C09100=1019.861,101.441,387.765,167.239,51.912,159.574
C09101=1019.866,101.689,387.746,167.241,51.905,159.573
C09102=1019.872,101.938,387.728,167.244,51.898,159.572
C09103=1019.877,102.188,387.710,167.246,51.892,159.571
C09104=1019.882,102.438,387.692,167.249,51.885,159.571
C09105=1019.888,102.686,387.673,167.252,51.878,159.570
C09106=1019.893,102.936,387.655,167.255,51.871,159.569
C09107=1019.898,103.185,387.637,167.257,51.864,159.568
C09108=1019.903,103.435,387.619,167.260,51.857,159.567
C09109=1019.910,103.684,387.601,167.263,51.851,159.567
C09110=1019.914,103.933,387.582,167.266,51.844,159.566
C09111=1019.919,104.182,387.564,167.269,51.838,159.565
C09112=1019.925,104.432,387.546,167.272,51.831,159.564
C09113=1019.930,104.681,387.527,167.274,51.824,159.563
C09114=1019.936,104.930,387.510,167.277,51.817,159.563
C09115=1019.941,105.180,387.491,167.280,51.811,159.562
C09116=1019.946,105.429,387.472,167.283,51.804,159.561
C09117=1019.952,105.678,387.455,167.285,51.797,159.560
C09118=1019.957,105.928,387.436,167.288,51.790,159.559
C09119=1019.963,106.176,387.418,167.292,51.783,159.559
C09120=1019.968,106.426,387.400,167.294,51.776,159.558
C09121=1019.974,106.675,387.382,167.297,51.769,159.557
C09122=1019.979,106.958,387.360,167.300,51.762,159.556
C09123=1019.986,107.241,387.340,167.303,51.754,159.555
C09124=1019.992,107.524,387.319,167.307,51.746,159.554
C09125=1019.998,107.806,387.298,167.310,51.738,159.553
C09126=1020.004,108.056,387.280,167.312,51.732,159.552
C09127=1020.009,108.305,387.262,167.315,51.725,159.551
C09128=1020.014,108.554,387.243,167.318,51.718,159.551
C09129=1020.020,108.804,387.225,167.321,51.711,159.550
C09130=1020.025,109.052,387.206,167.324,51.704,159.549
C09131=1020.032,109.302,387.188,167.326,51.698,159.548
C09132=1020.036,109.551,387.170,167.330,51.691,159.547
C09133=1020.041,109.800,387.151,167.332,51.684,159.546
C09134=1020.047,110.050,387.133,167.335,51.678,159.546
C09135=1020.053,110.299,387.115,167.338,51.671,159.545
C09136=1020.058,110.549,387.096,167.341,51.664,159.544
C09137=1020.063,110.797,387.077,167.344,51.657,159.543
C09138=1020.068,111.047,387.059,167.347,51.651,159.543
C09139=1020.074,111.296,387.040,167.350,51.644,159.542
C09140=1020.079,111.545,387.021,167.352,51.637,159.541
C09141=1020.085,111.795,387.003,167.355,51.630,159.540
C09142=1020.090,112.043,386.984,167.358,51.623,159.539
C09143=1020.095,112.293,386.966,167.361,51.616,159.539
C09144=1020.100,112.542,386.947,167.363,51.610,159.538
C09145=1020.106,112.792,386.927,167.367,51.603,159.537
C09146=1020.111,113.041,386.909,167.369,51.597,159.536
C09147=1020.116,113.290,386.890,167.373,51.590,159.535
C09148=1020.122,113.539,386.871,167.375,51.583,159.535
C09149=1020.127,113.789,386.853,167.378,51.576,159.534
C09150=1020.132,114.038,386.834,167.380,51.570,159.533
C09151=1020.137,114.287,386.815,167.384,51.564,159.532
C09152=1020.143,114.536,386.796,167.386,51.557,159.531
C09153=1020.148,114.785,386.777,167.390,51.550,159.531
C09154=1020.153,115.035,386.758,167.392,51.543,159.530
C09155=1020.158,115.284,386.739,167.395,51.536,159.529
C09156=1020.164,115.533,386.720,167.398,51.530,159.528
C09157=1020.169,115.782,386.702,167.401,51.523,159.527
C09158=1020.175,116.032,386.683,167.404,51.517,159.527
C09159=1020.179,116.281,386.663,167.407,51.510,159.526
C09160=1020.185,116.530,386.644,167.409,51.504,159.525
C09161=1020.190,116.779,386.625,167.412,51.497,159.524
C09162=1020.195,117.029,386.607,167.415,51.490,159.523
C09163=1020.200,117.278,386.588,167.418,51.483,159.523
C09164=1020.206,117.527,386.568,167.421,51.476,159.522
C09165=1020.211,117.776,386.550,167.424,51.470,159.521
C09166=1020.217,118.025,386.530,167.427,51.463,159.520
C09167=1020.222,118.274,386.511,167.430,51.457,159.520
C09168=1020.227,118.524,386.493,167.433,51.450,159.519
C09169=1020.232,118.773,386.474,167.435,51.443,159.518
C09170=1020.238,119.022,386.455,167.439,51.436,159.517
C09171=1020.243,119.271,386.436,167.441,51.430,159.516
C09172=1020.249,119.521,386.417,167.444,51.423,159.516
C09173=1020.254,119.770,386.397,167.448,51.416,159.515
C09174=1020.259,120.019,386.378,167.450,51.409,159.514
C09175=1020.264,120.268,386.359,167.454,51.403,159.513
C09176=1020.269,120.517,386.340,167.456,51.396,159.512
C09177=1020.275,120.767,386.321,167.459,51.390,159.512
C09178=1020.280,121.016,386.302,167.463,51.383,159.511
C09179=1020.286,121.265,386.283,167.465,51.376,159.510
C09180=1020.291,121.515,386.264,167.468,51.369,159.509
C09181=1020.296,121.764,386.245,167.471,51.363,159.508
C09182=1020.302,122.013,386.226,167.474,51.356,159.508
C09183=1020.307,122.262,386.207,167.477,51.349,159.507
C09184=1020.313,122.511,386.188,167.480,51.342,159.506
C09185=1020.318,122.761,386.168,167.483,51.335,159.505
C09186=1020.324,123.043,386.147,167.486,51.328,159.504
C09187=1020.330,123.326,386.125,167.490,51.320,159.503
C09188=1020.336,123.609,386.103,167.493,51.312,159.502
C09189=1020.342,123.891,386.082,167.496,51.305,159.502
C09190=1020.348,124.141,386.062,167.499,51.298,159.501
C09191=1020.353,124.389,386.043,167.503,51.291,159.500
C09192=1020.359,124.639,386.024,167.505,51.285,159.499
C09193=1020.364,124.889,386.004,167.508,51.278,159.498
C09194=1020.369,125.137,385.985,167.512,51.271,159.498
C09195=1020.375,125.387,385.966,167.514,51.264,159.497
C09196=1020.380,125.636,385.947,167.517,51.257,159.496
C09197=1020.385,125.885,385.928,167.520,51.251,159.495
C09198=1020.391,126.134,385.909,167.523,51.244,159.494
C09199=1020.397,126.384,385.890,167.526,51.237,159.494
C09200=1020.402,126.633,385.871,167.530,51.230,159.493
C09201=1020.408,126.882,385.852,167.532,51.224,159.492
C09202=1020.413,127.131,385.832,167.536,51.217,159.491
C09203=1020.418,127.380,385.812,167.539,51.210,159.490
C09204=1020.424,127.629,385.793,167.541,51.203,159.489
C09205=1020.429,127.879,385.774,167.544,51.196,159.489
C09206=1020.435,128.128,385.754,167.548,51.189,159.488
C09207=1020.440,128.377,385.735,167.550,51.182,159.487
C09208=1020.446,128.626,385.716,167.553,51.175,159.486
C09209=1020.451,128.876,385.697,167.557,51.169,159.485
C09210=1020.456,129.124,385.678,167.559,51.162,159.484
C09211=1020.462,129.374,385.659,167.562,51.155,159.484
C09212=1020.468,129.623,385.639,167.566,51.148,159.483
C09213=1020.473,129.872,385.619,167.569,51.141,159.482
C09214=1020.478,130.121,385.600,167.571,51.135,159.481
C09215=1020.484,130.371,385.581,167.575,51.128,159.481
C09216=1020.489,130.620,385.560,167.577,51.122,159.480
C09217=1020.495,130.869,385.541,167.581,51.115,159.479
C09218=1020.500,131.119,385.521,167.584,51.108,159.478
C09219=1020.505,131.368,385.502,167.587,51.102,159.477
C09220=1020.510,131.617,385.482,167.590,51.095,159.477
C09221=1020.516,131.866,385.463,167.593,51.088,159.476
C09222=1020.520,132.115,385.442,167.596,51.082,159.475
C09223=1020.526,132.364,385.423,167.599,51.075,159.474
C09224=1020.532,132.614,385.404,167.603,51.068,159.474
C09225=1020.537,132.863,385.383,167.605,51.062,159.473
C09226=1020.543,133.112,385.364,167.609,51.055,159.472
C09227=1020.547,133.361,385.345,167.611,51.049,159.471
C09228=1020.553,133.610,385.325,167.614,51.042,159.470
C09229=1020.558,133.860,385.305,167.618,51.035,159.470
C09230=1020.564,134.108,385.285,167.620,51.028,159.469
C09231=1020.568,134.358,385.265,167.623,51.021,159.468
C09232=1020.574,134.606,385.246,167.627,51.015,159.467
C09233=1020.579,134.856,385.226,167.630,51.008,159.466
C09234=1020.585,135.106,385.206,167.633,51.001,159.466
C09235=1020.591,135.354,385.186,167.636,50.995,159.465
C09236=1020.595,135.603,385.167,167.640,50.988,159.464
C09237=1020.601,135.852,385.147,167.642,50.982,159.463
C09238=1020.606,136.102,385.127,167.645,50.975,159.463
C09239=1020.612,136.351,385.107,167.649,50.968,159.462
C09240=1020.617,136.600,385.087,167.651,50.961,159.461
C09241=1020.623,136.850,385.067,167.655,50.955,159.460
C09242=1020.628,137.098,385.048,167.658,50.948,159.459
C09243=1020.633,137.347,385.027,167.660,50.941,159.459
C09244=1020.639,137.596,385.007,167.664,50.934,159.458
C09245=1020.644,137.846,384.988,167.668,50.928,159.457
C09246=1020.650,138.095,384.968,167.671,50.921,159.456
C09247=1020.655,138.345,384.948,167.673,50.915,159.456
C09248=1020.659,138.593,384.928,167.677,50.908,159.455
C09249=1020.665,138.842,384.908,167.680,50.901,159.454
C09250=1020.671,139.125,384.885,167.683,50.894,159.453
C09251=1020.677,139.408,384.862,167.687,50.887,159.452
C09252=1020.684,139.690,384.839,167.691,50.879,159.451
C09253=1020.689,139.973,384.816,167.694,50.871,159.450
C09254=1020.695,140.222,384.796,167.697,50.864,159.450
C09255=1020.700,140.472,384.776,167.701,50.858,159.449
C09256=1020.705,140.720,384.756,167.703,50.852,159.448
C09257=1020.710,140.969,384.736,167.707,50.845,159.447
C09258=1020.716,141.219,384.716,167.710,50.838,159.447
C09259=1020.721,141.468,384.696,167.712,50.832,159.446
C09260=1020.726,141.717,384.675,167.716,50.825,159.445
C09261=1020.732,141.966,384.655,167.719,50.818,159.444
C09262=1020.737,142.215,384.635,167.723,50.812,159.444
C09263=1020.743,142.464,384.615,167.725,50.805,159.443
C09264=1020.748,142.714,384.594,167.729,50.799,159.442
C09265=1020.754,142.962,384.574,167.732,50.792,159.441
C09266=1020.759,143.212,384.555,167.735,50.785,159.440
C09267=1020.763,143.461,384.534,167.738,50.778,159.440
C09268=1020.769,143.710,384.514,167.742,50.772,159.439
C09269=1020.775,143.959,384.494,167.745,50.765,159.438
C09270=1020.780,144.208,384.473,167.748,50.759,159.437
C09271=1020.785,144.457,384.453,167.751,50.752,159.437
C09272=1020.790,144.707,384.433,167.755,50.745,159.436
C09273=1020.796,144.955,384.413,167.758,50.738,159.435
C09274=1020.801,145.204,384.392,167.760,50.732,159.434
C09275=1020.807,145.454,384.372,167.764,50.725,159.433
C09276=1020.813,145.702,384.352,167.767,50.718,159.433
C09277=1020.818,145.952,384.331,167.771,50.712,159.432
C09278=1020.823,146.201,384.311,167.774,50.706,159.431
C09279=1020.828,146.450,384.290,167.777,50.699,159.430
C09280=1020.834,146.699,384.270,167.780,50.692,159.430
C09281=1020.839,146.949,384.250,167.784,50.685,159.429
C09282=1020.844,147.198,384.229,167.787,50.680,159.428
C09283=1020.849,147.447,384.209,167.790,50.673,159.427
C09284=1020.854,147.696,384.188,167.794,50.666,159.427
C09285=1020.860,147.945,384.168,167.797,50.659,159.426
C09286=1020.865,148.194,384.146,167.800,50.653,159.425
C09287=1020.870,148.443,384.126,167.803,50.647,159.424
C09288=1020.876,148.692,384.105,167.807,50.640,159.424
C09289=1020.881,148.941,384.085,167.810,50.633,159.423
C09290=1020.886,149.190,384.064,167.812,50.626,159.422
C09291=1020.891,149.439,384.044,167.816,50.620,159.421
C09292=1020.897,149.688,384.023,167.820,50.614,159.421
C09293=1020.902,149.938,384.002,167.823,50.607,159.420
C09294=1020.907,150.187,383.982,167.826,50.600,159.419
C09295=1020.912,150.436,383.961,167.829,50.594,159.418
C09296=1020.918,150.685,383.941,167.833,50.587,159.418
C09297=1020.923,150.934,383.920,167.836,50.581,159.417
C09298=1020.929,151.183,383.899,167.839,50.574,159.416
C09299=1020.934,151.432,383.878,167.842,50.567,159.415
C09300=1020.940,151.681,383.858,167.846,50.561,159.415
C09301=1020.945,151.931,383.837,167.850,50.554,159.414
C09302=1020.950,152.180,383.816,167.853,50.548,159.413
C09303=1020.955,152.429,383.796,167.855,50.541,159.412
C09304=1020.961,152.677,383.775,167.859,50.534,159.411
C09305=1020.966,152.926,383.754,167.863,50.528,159.411
C09306=1020.971,153.176,383.733,167.866,50.522,159.410
C09307=1020.977,153.425,383.713,167.870,50.515,159.409
C09308=1020.982,153.674,383.692,167.872,50.508,159.408
C09309=1020.988,153.923,383.671,167.876,50.502,159.408
C09310=1020.993,154.172,383.650,167.879,50.495,159.407
C09311=1020.999,154.421,383.630,167.883,50.489,159.406
C09312=1021.003,154.670,383.608,167.887,50.483,159.406
C09313=1021.009,154.919,383.587,167.889,50.476,159.405
C09314=1021.015,155.201,383.563,167.893,50.468,159.404
C09315=1021.021,155.484,383.540,167.897,50.462,159.403
C09316=1021.027,155.766,383.516,167.901,50.454,159.402
C09317=1021.033,156.050,383.493,167.905,50.446,159.402
C09318=1021.039,156.298,383.471,167.908,50.440,159.401
C09319=1021.043,156.548,383.450,167.911,50.433,159.400
C09320=1021.049,156.797,383.430,167.915,50.427,159.399
C09321=1021.054,157.045,383.408,167.918,50.420,159.399
C09322=1021.059,157.294,383.388,167.922,50.414,159.398
C09323=1021.066,157.543,383.366,167.926,50.407,159.397
C09324=1021.071,157.793,383.346,167.928,50.401,159.396
C09325=1021.075,158.042,383.324,167.931,50.394,159.396
C09326=1021.081,158.291,383.303,167.935,50.388,159.395
C09327=1021.086,158.540,383.283,167.939,50.381,159.394
C09328=1021.092,158.789,383.261,167.942,50.374,159.393
C09329=1021.098,159.038,383.240,167.946,50.368,159.393
C09330=1021.102,159.287,383.219,167.949,50.362,159.392
C09331=1021.107,159.536,383.197,167.952,50.356,159.391
C09332=1021.113,159.785,383.176,167.956,50.349,159.391
C09333=1021.117,160.034,383.154,167.959,50.342,159.390
C09334=1021.123,160.283,383.132,167.962,50.337,159.389
C09335=1021.128,160.532,383.112,167.966,50.330,159.388
C09336=1021.133,160.781,383.090,167.970,50.324,159.388
C09337=1021.138,161.030,383.068,167.973,50.317,159.387
C09338=1021.143,161.279,383.047,167.976,50.311,159.386
C09339=1021.148,161.528,383.025,167.979,50.304,159.386
C09340=1021.154,161.777,383.004,167.983,50.298,159.385
C09341=1021.159,162.026,382.982,167.987,50.292,159.384
C09342=1021.163,162.275,382.961,167.991,50.286,159.384
C09343=1021.169,162.524,382.939,167.993,50.279,159.383
C09344=1021.174,162.773,382.917,167.997,50.273,159.382
C09345=1021.180,163.022,382.896,168.000,50.266,159.381
C09346=1021.184,163.271,382.875,168.004,50.260,159.381
C09347=1021.189,163.520,382.853,168.008,50.254,159.380
C09348=1021.195,163.769,382.831,168.011,50.248,159.379
C09349=1021.200,164.018,382.809,168.014,50.241,159.379
C09350=1021.205,164.267,382.788,168.018,50.235,159.378
C09351=1021.211,164.517,382.767,168.022,50.228,159.377
C09352=1021.216,164.765,382.745,168.025,50.222,159.377
C09353=1021.221,165.014,382.723,168.028,50.216,159.376
C09354=1021.226,165.263,382.702,168.031,50.209,159.375
C09355=1021.231,165.512,382.679,168.035,50.203,159.374
C09356=1021.237,165.761,382.658,168.039,50.196,159.374
C09357=1021.242,166.010,382.637,168.043,50.190,159.373
C09358=1021.247,166.260,382.615,168.046,50.184,159.372
C09359=1021.253,166.508,382.594,168.050,50.178,159.372
C09360=1021.257,166.757,382.572,168.053,50.171,159.371
C09361=1021.263,167.007,382.549,168.056,50.165,159.370
C09362=1021.268,167.255,382.528,168.060,50.158,159.370
C09363=1021.273,167.504,382.506,168.064,50.152,159.369
C09364=1021.279,167.753,382.484,168.067,50.146,159.368
C09365=1021.284,168.002,382.463,168.071,50.140,159.368
C09366=1021.289,168.251,382.441,168.075,50.133,159.367
C09367=1021.294,168.500,382.419,168.078,50.126,159.366
C09368=1021.300,168.749,382.397,168.082,50.120,159.365
C09369=1021.305,168.998,382.376,168.085,50.114,159.365
C09370=1021.311,169.247,382.355,168.089,50.108,159.364
C09371=1021.315,169.496,382.333,168.092,50.101,159.363
C09372=1021.321,169.746,382.311,168.096,50.095,159.363
C09373=1021.326,169.994,382.289,168.100,50.088,159.362
C09374=1021.331,170.243,382.267,168.103,50.082,159.361
C09375=1021.337,170.493,382.245,168.107,50.076,159.360
C09376=1021.342,170.741,382.224,168.111,50.070,159.360
C09377=1021.348,170.990,382.201,168.114,50.063,159.359
C09378=1021.354,171.272,382.177,168.119,50.056,159.358
C09379=1021.360,171.554,382.151,168.122,50.048,159.357
C09380=1021.366,171.836,382.127,168.127,50.041,159.357
C09381=1021.372,172.118,382.102,168.131,50.034,159.356
C09382=1021.377,172.367,382.080,168.135,50.028,159.355
C09383=1021.383,172.617,382.058,168.138,50.021,159.355
C09384=1021.388,172.865,382.037,168.142,50.015,159.354
C09385=1021.394,173.115,382.015,168.146,50.008,159.353
C09386=1021.398,173.364,381.993,168.150,50.002,159.353
C09387=1021.405,173.613,381.971,168.153,49.996,159.352
C09388=1021.409,173.862,381.949,168.157,49.989,159.351
C09389=1021.415,174.111,381.926,168.161,49.983,159.350
C09390=1021.421,174.359,381.905,168.164,49.976,159.350
C09391=1021.426,174.609,381.883,168.168,49.970,159.349
C09392=1021.431,174.857,381.861,168.171,49.964,159.348
C09393=1021.437,175.107,381.839,168.175,49.957,159.348
C09394=1021.442,175.355,381.817,168.179,49.951,159.347
C09395=1021.448,175.604,381.795,168.183,49.945,159.346
C09396=1021.453,175.853,381.773,168.186,49.938,159.346
C09397=1021.459,176.102,381.751,168.190,49.931,159.345
C09398=1021.464,176.352,381.729,168.194,49.925,159.344
C09399=1021.470,176.600,381.707,168.197,49.919,159.343
C09400=1021.475,176.849,381.685,168.201,49.913,159.343
C09401=1021.480,177.098,381.663,168.205,49.906,159.342
C09402=1021.486,177.347,381.641,168.209,49.900,159.341
C09403=1021.492,177.595,381.619,168.212,49.893,159.341
C09404=1021.497,177.845,381.596,168.216,49.887,159.340
C09405=1021.502,178.095,381.574,168.220,49.881,159.339
C09406=1021.508,178.343,381.553,168.223,49.874,159.339
C09407=1021.514,178.592,381.530,168.227,49.868,159.338
C09408=1021.518,178.841,381.508,168.231,49.861,159.337
C09409=1021.525,179.090,381.486,168.236,49.855,159.337
C09410=1021.530,179.339,381.463,168.239,49.848,159.336
C09411=1021.535,179.588,381.442,168.243,49.842,159.335
C09412=1021.541,179.837,381.420,168.247,49.836,159.335
C09413=1021.547,180.086,381.397,168.251,49.830,159.334
C09414=1021.552,180.335,381.375,168.254,49.823,159.333
C09415=1021.558,180.584,381.353,168.258,49.817,159.333
C09416=1021.564,180.833,381.331,168.262,49.810,159.332
C09417=1021.569,181.081,381.309,168.265,49.804,159.331
C09418=1021.575,181.330,381.286,168.270,49.798,159.331
C09419=1021.581,181.580,381.264,168.274,49.791,159.330
C09420=1021.586,181.828,381.241,168.278,49.785,159.329
C09421=1021.591,182.077,381.219,168.281,49.778,159.328
C09422=1021.597,182.327,381.197,168.285,49.772,159.328
C09423=1021.602,182.575,381.174,168.289,49.766,159.327
C09424=1021.607,182.824,381.152,168.293,49.760,159.326
C09425=1021.612,183.074,381.129,168.297,49.754,159.326
C09426=1021.618,183.323,381.106,168.301,49.748,159.325
C09427=1021.623,183.571,381.083,168.305,49.742,159.325
C09428=1021.628,183.820,381.060,168.308,49.736,159.324
C09429=1021.633,184.070,381.037,168.312,49.729,159.323
C09430=1021.638,184.318,381.015,168.316,49.723,159.323
C09431=1021.644,184.567,380.992,168.320,49.717,159.322
C09432=1021.649,184.816,380.968,168.324,49.711,159.322
C09433=1021.654,185.064,380.946,168.327,49.705,159.321
C09434=1021.660,185.314,380.924,168.331,49.699,159.320
C09435=1021.665,185.563,380.900,168.335,49.693,159.320
C09436=1021.670,185.811,380.877,168.339,49.687,159.319
C09437=1021.676,186.060,380.854,168.343,49.681,159.318
C09438=1021.681,186.309,380.831,168.347,49.674,159.318
C09439=1021.686,186.558,380.808,168.351,49.668,159.317
C09440=1021.691,186.806,380.785,168.355,49.662,159.316
C09441=1021.696,187.056,380.763,168.359,49.656,159.316
C09442=1021.702,187.338,380.736,168.363,49.649,159.315
C09443=1021.708,187.619,380.710,168.368,49.642,159.314
C09444=1021.714,187.901,380.684,168.372,49.635,159.314
C09445=1021.720,188.183,380.658,168.377,49.628,159.313
C09446=1021.726,188.431,380.636,168.381,49.622,159.312
C09447=1021.731,188.680,380.613,168.385,49.616,159.312
C09448=1021.736,188.929,380.589,168.388,49.610,159.311
C09449=1021.742,189.178,380.566,168.392,49.604,159.310
C09450=1021.748,189.427,380.543,168.396,49.598,159.310
C09451=1021.752,189.676,380.520,168.401,49.591,159.309
C09452=1021.758,189.924,380.497,168.405,49.585,159.309
C09453=1021.764,190.173,380.474,168.409,49.579,159.308
C09454=1021.769,190.423,380.451,168.413,49.573,159.307
C09455=1021.774,190.671,380.428,168.417,49.567,159.307
C09456=1021.780,190.920,380.405,168.420,49.561,159.306
C09457=1021.784,191.169,380.381,168.424,49.555,159.305
C09458=1021.790,191.418,380.359,168.429,49.549,159.305
C09459=1021.796,191.667,380.336,168.433,49.543,159.304
C09460=1021.801,191.916,380.312,168.437,49.537,159.304
C09461=1021.807,192.165,380.289,168.441,49.531,159.303
C09462=1021.813,192.413,380.265,168.445,49.524,159.302
C09463=1021.818,192.662,380.242,168.449,49.518,159.302
C09464=1021.823,192.911,380.219,168.454,49.512,159.301
C09465=1021.828,193.160,380.196,168.458,49.506,159.301
C09466=1021.834,193.409,380.173,168.462,49.500,159.300
C09467=1021.839,193.657,380.150,168.465,49.493,159.299
C09468=1021.844,193.907,380.126,168.469,49.488,159.299
C09469=1021.850,194.156,380.103,168.474,49.481,159.298
C09470=1021.856,194.404,380.080,168.478,49.475,159.298
C09471=1021.861,194.653,380.056,168.482,49.469,159.297
C09472=1021.867,194.902,380.033,168.486,49.464,159.296
C09473=1021.872,195.151,380.010,168.490,49.457,159.296
C09474=1021.877,195.400,379.987,168.495,49.451,159.295
C09475=1021.883,195.648,379.963,168.499,49.445,159.295
C09476=1021.889,195.897,379.940,168.503,49.439,159.294
C09477=1021.894,196.146,379.917,168.507,49.433,159.293
C09478=1021.900,196.395,379.894,168.512,49.427,159.293
C09479=1021.905,196.644,379.869,168.516,49.421,159.292
C09480=1021.911,196.893,379.846,168.519,49.414,159.291
C09481=1021.917,197.142,379.824,168.523,49.408,159.291
C09482=1021.922,197.390,379.799,168.528,49.402,159.290
C09483=1021.928,197.639,379.776,168.532,49.396,159.290
C09484=1021.933,197.888,379.753,168.536,49.390,159.289
C09485=1021.939,198.137,379.729,168.540,49.384,159.289
C09486=1021.944,198.386,379.706,168.545,49.378,159.288
C09487=1021.950,198.634,379.683,168.549,49.372,159.287
C09488=1021.956,198.883,379.659,168.553,49.366,159.287
C09489=1021.961,199.132,379.636,168.558,49.359,159.286
C09490=1021.966,199.381,379.613,168.562,49.354,159.286
C09491=1021.972,199.629,379.589,168.566,49.348,159.285
C09492=1021.977,199.879,379.565,168.571,49.341,159.284
C09493=1021.984,200.128,379.541,168.575,49.336,159.284
C09494=1021.989,200.377,379.518,168.579,49.330,159.283
C09495=1021.994,200.625,379.493,168.583,49.324,159.283
C09496=1021.999,200.874,379.469,168.586,49.318,159.282
C09497=1022.005,201.123,379.446,168.591,49.312,159.281
C09498=1022.011,201.371,379.422,168.595,49.306,159.281
C09499=1022.016,201.621,379.398,168.599,49.300,159.280
C09500=1022.021,201.869,379.374,168.604,49.294,159.280
C09501=1022.027,202.118,379.351,168.608,49.288,159.279
C09502=1022.032,202.367,379.327,168.613,49.283,159.279
C09503=1022.037,202.615,379.303,168.617,49.277,159.278
C09504=1022.043,202.865,379.278,168.622,49.270,159.278
C09505=1022.049,203.114,379.255,168.626,49.265,159.277
C09506=1022.077,204.361,379.134,169.059,49.356,159.363
C09507=1022.082,204.574,379.111,169.061,49.352,159.363
C09508=1022.088,204.787,379.090,169.065,49.348,159.363
C09509=1022.093,205.000,379.068,169.067,49.343,159.362
C09510=1022.099,205.213,379.046,169.071,49.339,159.362
C09511=1022.104,205.425,379.025,169.073,49.334,159.361
C09512=1022.109,205.639,379.002,169.077,49.330,159.361
C09513=1022.115,205.852,378.981,169.079,49.326,159.360
C09514=1022.121,206.100,378.955,169.083,49.321,159.360
C09515=1022.128,206.349,378.929,169.086,49.317,159.359
C09516=1022.134,206.598,378.904,169.089,49.312,159.359
C09517=1022.141,206.846,378.878,169.093,49.307,159.358
C09518=1022.147,207.095,378.853,169.096,49.302,159.358
C09519=1022.153,207.343,378.827,169.100,49.297,159.357
C09520=1022.159,207.592,378.802,169.103,49.292,159.357
C09521=1022.166,207.840,378.776,169.107,49.287,159.356
C09522=1022.171,208.089,378.750,169.110,49.282,159.356
C09523=1022.178,208.339,378.724,169.113,49.277,159.355
C09524=1022.185,208.587,378.698,169.117,49.272,159.355
C09525=1022.191,208.835,378.673,169.120,49.267,159.354
C09526=1022.197,209.083,378.647,169.123,49.262,159.353
C09527=1022.203,209.332,378.621,169.127,49.258,159.353
C09528=1022.210,209.581,378.596,169.130,49.253,159.352
C09529=1022.216,209.830,378.569,169.134,49.248,159.352
C09530=1022.222,210.078,378.544,169.138,49.243,159.352
C09531=1022.229,210.326,378.518,169.141,49.238,159.351
C09532=1022.235,210.575,378.492,169.144,49.234,159.351
C09533=1022.241,210.823,378.466,169.148,49.229,159.350
C09534=1022.247,211.072,378.440,169.151,49.224,159.349
C09535=1022.254,211.321,378.414,169.155,49.220,159.349
C09536=1022.260,211.570,378.388,169.158,49.215,159.349
C09537=1022.266,211.818,378.362,169.161,49.210,159.348
C09538=1022.272,212.067,378.337,169.164,49.205,159.348
C09539=1022.278,212.315,378.310,169.168,49.201,159.347
C09540=1022.285,212.564,378.284,169.171,49.196,159.347
C09541=1022.291,212.812,378.258,169.175,49.191,159.346
C09542=1022.297,213.061,378.232,169.178,49.187,159.346
C09543=1022.303,213.309,378.206,169.182,49.182,159.345
C09544=1022.310,213.558,378.180,169.185,49.177,159.345
C09545=1022.316,213.807,378.154,169.190,49.172,159.344
C09546=1022.322,214.055,378.128,169.193,49.168,159.344
C09547=1022.329,214.303,378.102,169.196,49.163,159.343
C09548=1022.335,214.553,378.076,169.200,49.158,159.343
C09549=1022.342,214.801,378.049,169.203,49.154,159.343
C09550=1022.348,215.049,378.023,169.206,49.149,159.342
C09551=1022.354,215.299,377.997,169.210,49.145,159.342
C09552=1022.361,215.547,377.971,169.213,49.140,159.341
C09553=1022.367,215.795,377.945,169.217,49.135,159.341
C09554=1022.373,216.044,377.919,169.220,49.131,159.340
C09555=1022.380,216.292,377.893,169.224,49.126,159.340
C09556=1022.386,216.541,377.867,169.227,49.121,159.339
C09557=1022.392,216.789,377.840,169.231,49.117,159.339
C09558=1022.399,217.038,377.814,169.234,49.112,159.338
C09559=1022.405,217.287,377.788,169.238,49.108,159.338
C09560=1022.411,217.535,377.762,169.241,49.103,159.337
C09561=1022.418,217.783,377.735,169.245,49.098,159.337
C09562=1022.424,218.032,377.709,169.249,49.093,159.337
C09563=1022.430,218.280,377.683,169.252,49.089,159.336
C09564=1022.437,218.529,377.657,169.256,49.084,159.336
C09565=1022.443,218.778,377.630,169.259,49.080,159.335
C09566=1022.449,218.993,377.607,169.262,49.076,159.335
C09567=1022.454,219.207,377.585,169.265,49.072,159.334
C09568=1022.460,219.422,377.561,169.269,49.068,159.334
C09569=1022.464,219.637,377.538,169.271,49.064,159.334
C09570=1022.470,219.852,377.516,169.274,49.060,159.333
C09571=1022.475,220.067,377.493,169.278,49.057,159.333
C09572=1022.481,220.281,377.470,169.280,49.053,159.333
C09573=1022.486,220.496,377.447,169.283,49.049,159.332
C09574=1022.493,220.745,377.420,169.287,49.045,159.332
C09575=1022.499,220.993,377.394,169.290,49.040,159.331
C09576=1022.505,221.241,377.367,169.294,49.036,159.331
C09577=1022.512,221.490,377.341,169.297,49.032,159.331
C09578=1022.517,221.739,377.314,169.301,49.027,159.330
C09579=1022.525,221.987,377.288,169.304,49.023,159.330
C09580=1022.530,222.236,377.261,169.308,49.018,159.329
C09581=1022.536,222.484,377.234,169.311,49.014,159.329
C09582=1022.543,222.733,377.208,169.315,49.009,159.329
C09583=1022.549,222.981,377.181,169.319,49.005,159.328
C09584=1022.555,223.230,377.154,169.322,49.000,159.328
C09585=1022.562,223.478,377.128,169.326,48.996,159.327
C09586=1022.568,223.727,377.101,169.329,48.992,159.327
C09587=1022.574,223.975,377.074,169.333,48.988,159.327
C09588=1022.581,224.224,377.047,169.336,48.983,159.326
C09589=1022.587,224.472,377.021,169.340,48.979,159.326
C09590=1022.593,224.721,376.994,169.344,48.975,159.325
C09591=1022.600,224.969,376.968,169.347,48.970,159.325
C09592=1022.606,225.218,376.941,169.351,48.966,159.324
C09593=1022.612,225.467,376.914,169.354,48.961,159.324
C09594=1022.619,225.714,376.887,169.358,48.957,159.324
C09595=1022.625,225.963,376.860,169.362,48.953,159.323
C09596=1022.631,226.212,376.834,169.366,48.949,159.323
C09597=1022.638,226.460,376.807,169.370,48.944,159.323
C09598=1022.644,226.709,376.780,169.373,48.940,159.322
C09599=1022.652,226.957,376.753,169.377,48.935,159.322
C09600=1022.657,227.205,376.727,169.381,48.931,159.322
C09601=1022.664,227.454,376.700,169.383,48.927,159.321
C09602=1022.670,227.702,376.672,169.387,48.923,159.321
C09603=1022.676,227.951,376.645,169.391,48.919,159.320
C09604=1022.682,228.199,376.619,169.394,48.915,159.320
C09605=1022.689,228.448,376.591,169.398,48.911,159.320
C09606=1022.695,228.697,376.564,169.402,48.907,159.319
C09607=1022.701,228.945,376.537,169.405,48.902,159.319
C09608=1022.707,229.194,376.510,169.409,48.898,159.319
C09609=1022.714,229.442,376.483,169.413,48.894,159.318
C09610=1022.721,229.690,376.456,169.416,48.890,159.318
C09611=1022.726,229.939,376.429,169.420,48.886,159.318
C09612=1022.733,230.188,376.402,169.424,48.882,159.317
C09613=1022.739,230.435,376.375,169.427,48.877,159.317
C09614=1022.745,230.684,376.348,169.431,48.873,159.317
C09615=1022.752,230.933,376.320,169.435,48.869,159.316
C09616=1022.758,231.181,376.293,169.438,48.865,159.316
C09617=1022.764,231.430,376.266,169.442,48.861,159.315
C09618=1022.770,231.677,376.238,169.446,48.857,159.315
C09619=1022.777,231.926,376.211,169.449,48.852,159.315
C09620=1022.783,232.175,376.183,169.453,48.849,159.315
C09621=1022.789,232.423,376.157,169.457,48.845,159.314
C09622=1022.795,232.672,376.128,169.461,48.841,159.314
C09623=1022.801,232.920,376.102,169.465,48.836,159.314
C09624=1022.808,233.169,376.074,169.468,48.832,159.313
C09625=1022.814,233.417,376.046,169.471,48.828,159.313
C09626=1022.824,233.793,376.006,169.477,48.823,159.312
C09627=1022.834,234.169,375.964,169.482,48.817,159.312
C09628=1022.843,234.546,375.923,169.488,48.810,159.311
C09629=1022.853,234.922,375.881,169.494,48.805,159.311
C09630=1022.859,235.170,375.854,169.497,48.801,159.311
C09631=1022.865,235.419,375.826,169.501,48.796,159.310
C09632=1022.872,235.667,375.799,169.505,48.792,159.310
C09633=1022.878,235.915,375.771,169.509,48.789,159.310
C09634=1022.884,236.165,375.744,169.512,48.785,159.309
C09635=1022.891,236.413,375.716,169.516,48.780,159.309
C09636=1022.897,236.661,375.689,169.520,48.776,159.309
C09637=1022.903,236.909,375.661,169.524,48.773,159.309
C09638=1022.910,237.158,375.633,169.527,48.769,159.308
C09639=1022.916,237.407,375.606,169.531,48.765,159.308
C09640=1022.922,237.654,375.579,169.535,48.761,159.308
C09641=1022.929,237.903,375.551,169.539,48.757,159.307
C09642=1022.935,238.152,375.523,169.543,48.753,159.307
C09643=1022.942,238.400,375.495,169.547,48.749,159.307
C09644=1022.948,238.648,375.468,169.550,48.745,159.306
C09645=1022.954,238.897,375.441,169.554,48.741,159.306
C09646=1022.961,239.145,375.413,169.558,48.737,159.306
C09647=1022.968,239.394,375.385,169.562,48.733,159.306
C09648=1022.973,239.642,375.357,169.566,48.730,159.305
C09649=1022.980,239.890,375.330,169.569,48.726,159.305
C09650=1022.986,240.139,375.302,169.572,48.722,159.305
C09651=1022.992,240.387,375.273,169.576,48.718,159.304
C09652=1022.998,240.635,375.246,169.580,48.715,159.304
C09653=1023.004,240.884,375.218,169.584,48.711,159.304
C09654=1023.011,241.132,375.190,169.588,48.707,159.304
C09655=1023.018,241.380,375.162,169.592,48.704,159.304
C09656=1023.023,241.628,375.134,169.595,48.700,159.303
C09657=1023.030,241.877,375.106,169.600,48.696,159.303
C09658=1023.036,242.125,375.078,169.603,48.692,159.303
C09659=1023.043,242.374,375.050,169.607,48.689,159.303
C09660=1023.049,242.622,375.022,169.611,48.684,159.302
C09661=1023.055,242.871,374.994,169.614,48.681,159.302
C09662=1023.061,243.119,374.966,169.618,48.678,159.302
C09663=1023.068,243.367,374.937,169.622,48.674,159.301
C09664=1023.074,243.615,374.910,169.626,48.670,159.301
C09665=1023.080,243.864,374.881,169.630,48.667,159.301
C09666=1023.087,244.113,374.854,169.633,48.662,159.301
C09667=1023.092,244.360,374.825,169.637,48.659,159.301
C09668=1023.098,244.609,374.797,169.641,48.656,159.300
C09669=1023.105,244.857,374.769,169.646,48.652,159.300
C09670=1023.111,245.105,374.740,169.649,48.649,159.300
C09671=1023.117,245.354,374.712,169.652,48.645,159.300
C09672=1023.124,245.602,374.684,169.656,48.641,159.299
C09673=1023.130,245.850,374.655,169.660,48.638,159.299
C09674=1023.136,246.099,374.627,169.664,48.634,159.299
C09675=1023.143,246.346,374.598,169.668,48.631,159.299
C09676=1023.149,246.595,374.570,169.672,48.627,159.299
C09677=1023.154,246.844,374.542,169.676,48.623,159.298
C09678=1023.162,247.138,374.508,169.680,48.620,159.298
C09679=1023.170,247.432,374.475,169.685,48.615,159.298
C09680=1023.177,247.726,374.441,169.690,48.611,159.298
C09681=1023.184,248.019,374.407,169.694,48.606,159.297
C09682=1023.195,248.434,374.359,169.701,48.601,159.297
C09683=1023.206,248.849,374.312,169.707,48.595,159.297
C09684=1023.216,249.265,374.264,169.713,48.589,159.296
C09685=1023.226,249.680,374.216,169.720,48.584,159.296
C09686=1023.233,249.928,374.188,169.724,48.580,159.296
C09687=1023.239,250.177,374.160,169.728,48.577,159.296
C09688=1023.245,250.425,374.131,169.732,48.573,159.296
C09689=1023.251,250.674,374.102,169.736,48.570,159.295
C09690=1023.258,250.922,374.074,169.740,48.566,159.295
C09691=1023.264,251.170,374.046,169.744,48.563,159.295
C09692=1023.270,251.418,374.017,169.748,48.559,159.295
C09693=1023.277,251.666,373.988,169.752,48.556,159.295
C09694=1023.283,251.915,373.960,169.756,48.553,159.295
C09695=1023.290,252.163,373.931,169.760,48.549,159.294
C09696=1023.296,252.411,373.902,169.763,48.546,159.294
C09697=1023.303,252.660,373.874,169.767,48.542,159.294
C09698=1023.309,252.908,373.845,169.771,48.539,159.294
C09699=1023.316,253.157,373.815,169.775,48.536,159.294
C09700=1023.322,253.405,373.788,169.779,48.532,159.293
C09701=1023.329,253.653,373.759,169.783,48.529,159.293
C09702=1023.335,253.901,373.730,169.787,48.525,159.293
C09703=1023.342,254.149,373.701,169.791,48.522,159.293
C09704=1023.348,254.398,373.673,169.795,48.518,159.293
C09705=1023.354,254.646,373.644,169.799,48.515,159.293
C09706=1023.360,254.894,373.615,169.804,48.511,159.292
C09707=1023.367,255.142,373.586,169.808,48.508,159.292
C09708=1023.373,255.391,373.558,169.812,48.505,159.292
C09709=1023.380,255.640,373.529,169.816,48.502,159.292
C09710=1023.387,255.887,373.500,169.819,48.498,159.292
C09711=1023.393,256.136,373.471,169.823,48.495,159.292
C09712=1023.400,256.384,373.442,169.827,48.491,159.291
C09713=1023.406,256.632,373.413,169.831,48.488,159.291
C09714=1023.413,256.880,373.385,169.835,48.485,159.291
C09715=1023.419,257.129,373.356,169.840,48.482,159.291
C09716=1023.426,257.377,373.327,169.844,48.478,159.291
C09717=1023.432,257.625,373.298,169.848,48.475,159.291
C09718=1023.439,257.873,373.269,169.852,48.471,159.291
C09719=1023.445,258.121,373.240,169.856,48.468,159.290
C09720=1023.452,258.370,373.211,169.860,48.465,159.290
C09721=1023.459,258.618,373.183,169.864,48.462,159.290
C09722=1023.465,258.866,373.153,169.868,48.458,159.290
C09723=1023.471,259.114,373.124,169.872,48.455,159.290
C09724=1023.478,259.363,373.095,169.877,48.452,159.290
C09725=1023.485,259.611,373.067,169.881,48.449,159.290
C09726=1023.492,259.859,373.038,169.885,48.445,159.289
C09727=1023.498,260.107,373.009,169.889,48.442,159.289
C09728=1023.505,260.355,372.980,169.893,48.439,159.289
C09729=1023.512,260.604,372.951,169.897,48.435,159.289
C09730=1023.518,260.852,372.922,169.901,48.433,159.289
C09731=1023.523,261.100,372.892,169.904,48.429,159.289
C09732=1023.530,261.348,372.862,169.909,48.427,159.289
C09733=1023.537,261.597,372.833,169.913,48.423,159.289
C09734=1023.543,261.845,372.804,169.917,48.420,159.289
C09735=1023.549,262.093,372.775,169.921,48.417,159.289
C09736=1023.556,262.341,372.745,169.926,48.414,159.289
C09737=1023.563,262.589,372.716,169.930,48.411,159.288
C09738=1023.573,263.003,372.666,169.936,48.406,159.288
C09739=1023.584,263.417,372.618,169.943,48.401,159.288
C09740=1023.595,263.831,372.568,169.950,48.396,159.288
C09741=1023.605,264.245,372.519,169.958,48.390,159.288
C09742=1023.612,264.493,372.490,169.961,48.387,159.288
C09743=1023.618,264.741,372.460,169.965,48.385,159.288
C09744=1023.624,264.990,372.430,169.970,48.382,159.288
C09745=1023.631,265.237,372.400,169.974,48.378,159.287
C09746=1023.637,265.485,372.371,169.978,48.375,159.287
C09747=1023.644,265.734,372.341,169.982,48.373,159.287
C09748=1023.651,265.982,372.312,169.986,48.369,159.287
C09749=1023.656,266.229,372.282,169.991,48.366,159.287
C09750=1023.663,266.478,372.253,169.995,48.364,159.287
C09751=1023.670,266.726,372.223,169.999,48.360,159.287
C09752=1023.676,266.975,372.193,170.004,48.357,159.287
C09753=1023.682,267.222,372.163,170.008,48.355,159.287
C09754=1023.689,267.471,372.134,170.011,48.352,159.287
C09755=1023.696,267.719,372.104,170.015,48.349,159.287
C09756=1023.702,267.967,372.073,170.020,48.346,159.287
C09757=1023.709,268.215,372.044,170.024,48.343,159.287
C09758=1023.715,268.463,372.014,170.028,48.340,159.287
C09759=1023.721,268.711,371.985,170.033,48.338,159.287
C09760=1023.728,268.960,371.955,170.037,48.334,159.287
C09761=1023.734,269.207,371.925,170.041,48.331,159.287
C09762=1023.741,269.456,371.894,170.046,48.329,159.287
C09763=1023.747,269.704,371.865,170.050,48.326,159.287
C09764=1023.754,269.952,371.835,170.054,48.323,159.287
C09765=1023.760,270.200,371.805,170.059,48.320,159.287
C09766=1023.767,270.447,371.775,170.063,48.317,159.287
C09767=1023.773,270.696,371.745,170.067,48.315,159.287
C09768=1023.779,270.944,371.715,170.071,48.312,159.287
C09769=1023.786,271.193,371.684,170.075,48.309,159.286
C09770=1023.792,271.440,371.655,170.079,48.306,159.286
C09771=1023.799,271.689,371.624,170.084,48.303,159.286
C09772=1023.805,271.936,371.594,170.088,48.300,159.286
C09773=1023.811,272.185,371.564,170.092,48.298,159.286
C09774=1023.818,272.433,371.534,170.097,48.295,159.286
C09775=1023.825,272.681,371.504,170.101,48.292,159.286
C09776=1023.831,272.929,371.474,170.106,48.289,159.286
C09777=1023.837,273.177,371.443,170.110,48.286,159.286
C09778=1023.844,273.425,371.413,170.115,48.284,159.287
C09779=1023.850,273.673,371.383,170.118,48.282,159.287
C09780=1023.857,273.922,371.353,170.122,48.279,159.287
C09781=1023.863,274.169,371.322,170.127,48.276,159.287
C09782=1023.870,274.418,371.292,170.131,48.274,159.287
C09783=1023.876,274.665,371.262,170.136,48.271,159.287
C09784=1023.883,274.914,371.232,170.140,48.268,159.287
C09785=1023.889,275.161,371.201,170.144,48.265,159.287
C09786=1023.896,275.409,371.170,170.149,48.262,159.287
C09787=1023.903,275.658,371.140,170.153,48.260,159.287
C09788=1023.909,275.905,371.109,170.158,48.258,159.287
C09789=1023.916,276.154,371.079,170.162,48.255,159.287
C09790=1023.922,276.401,371.049,170.167,48.252,159.287
C09791=1023.929,276.650,371.019,170.171,48.249,159.287
C09792=1023.935,276.898,370.988,170.175,48.246,159.287
C09793=1023.941,277.145,370.957,170.180,48.244,159.287
C09794=1023.953,277.564,370.906,170.187,48.240,159.287
C09795=1023.964,277.983,370.854,170.194,48.236,159.287
C09796=1023.974,278.401,370.802,170.201,48.231,159.287
C09797=1023.986,278.820,370.750,170.209,48.227,159.287
C09798=1023.992,279.067,370.720,170.214,48.225,159.287
C09799=1023.998,279.315,370.688,170.218,48.222,159.287
C09800=1024.005,279.564,370.658,170.223,48.220,159.288
C09801=1024.011,279.811,370.628,170.228,48.217,159.288
C09802=1024.018,280.059,370.596,170.231,48.214,159.287
C09803=1024.024,280.308,370.566,170.236,48.212,159.288
C09804=1024.030,280.555,370.535,170.240,48.210,159.288
C09805=1024.037,280.803,370.504,170.245,48.207,159.288
C09806=1024.044,281.051,370.473,170.249,48.205,159.288
C09807=1024.051,281.300,370.442,170.254,48.203,159.288
C09808=1024.057,281.547,370.411,170.258,48.200,159.288
C09809=1024.063,281.795,370.381,170.263,48.197,159.288
C09810=1024.070,282.043,370.349,170.267,48.195,159.288
C09811=1024.076,282.292,370.318,170.272,48.192,159.288
C09812=1024.083,282.539,370.287,170.276,48.190,159.288
C09813=1024.090,282.787,370.257,170.281,48.187,159.288
C09814=1024.096,283.035,370.226,170.286,48.185,159.289
C09815=1024.103,283.283,370.194,170.290,48.183,159.289
C09816=1024.110,283.532,370.164,170.295,48.180,159.289
C09817=1024.116,283.779,370.132,170.299,48.178,159.289
C09818=1024.122,284.027,370.102,170.304,48.175,159.289
C09819=1024.130,284.275,370.071,170.308,48.173,159.289
C09820=1024.136,284.523,370.040,170.313,48.170,159.289
C09821=1024.143,284.771,370.009,170.317,48.168,159.289
C09822=1024.149,285.019,369.977,170.322,48.166,159.289
C09823=1024.156,285.267,369.946,170.327,48.163,159.289
C09824=1024.162,285.514,369.915,170.331,48.161,159.290
C09825=1024.169,285.763,369.884,170.336,48.159,159.290
C09826=1024.175,286.011,369.853,170.340,48.156,159.290
C09827=1024.182,286.259,369.821,170.345,48.154,159.290
C09828=1024.189,286.506,369.790,170.350,48.152,159.290
C09829=1024.196,286.754,369.759,170.354,48.149,159.290
C09830=1024.202,287.002,369.727,170.359,48.147,159.290
C09831=1024.209,287.250,369.696,170.364,48.145,159.291
C09832=1024.216,287.498,369.664,170.368,48.143,159.291
C09833=1024.222,287.745,369.633,170.373,48.141,159.291
C09834=1024.228,287.994,369.602,170.377,48.138,159.291
C09835=1024.235,288.242,369.571,170.381,48.136,159.291
C09836=1024.242,288.490,369.540,170.386,48.134,159.291
C09837=1024.248,288.738,369.508,170.391,48.132,159.291
C09838=1024.255,288.985,369.475,170.395,48.130,159.292
C09839=1024.262,289.233,369.444,170.400,48.128,159.292
C09840=1024.268,289.481,369.413,170.405,48.126,159.292
C09841=1024.275,289.729,369.381,170.409,48.123,159.292
C09842=1024.282,289.977,369.350,170.414,48.121,159.292
C09843=1024.288,290.225,369.318,170.419,48.119,159.292
C09844=1024.294,290.473,369.286,170.423,48.117,159.292
C09845=1024.301,290.721,369.255,170.428,48.115,159.293
C09846=1024.308,290.969,369.223,170.433,48.112,159.293
C09847=1024.315,291.217,369.192,170.437,48.110,159.293
C09848=1024.322,291.464,369.160,170.442,48.108,159.293
C09849=1024.328,291.712,369.128,170.447,48.106,159.293
C09850=1024.334,291.927,369.101,170.451,48.104,159.293
C09851=1024.340,292.143,369.072,170.455,48.102,159.294
C09852=1024.345,292.358,369.045,170.460,48.101,159.294
C09853=1024.351,292.574,369.018,170.464,48.099,159.294
C09854=1024.357,292.788,368.990,170.468,48.097,159.294
C09855=1024.363,293.004,368.963,170.472,48.095,159.294
C09856=1024.368,293.219,368.934,170.476,48.093,159.294
C09857=1024.374,293.435,368.907,170.480,48.092,159.295
C09858=1024.381,293.682,368.875,170.485,48.090,159.295
C09859=1024.388,293.930,368.844,170.490,48.088,159.295
C09860=1024.394,294.178,368.811,170.494,48.086,159.295
C09861=1024.400,294.426,368.779,170.499,48.083,159.295
C09862=1024.407,294.673,368.747,170.504,48.082,159.296
C09863=1024.414,294.922,368.714,170.509,48.080,159.296
C09864=1024.421,295.169,368.682,170.513,48.078,159.296
C09865=1024.427,295.418,368.650,170.518,48.076,159.297
C09866=1024.433,295.665,368.617,170.523,48.074,159.297
C09867=1024.440,295.913,368.585,170.528,48.072,159.297
C09868=1024.446,296.161,368.553,170.533,48.071,159.297
C09869=1024.452,296.408,368.520,170.538,48.068,159.297
C09870=1024.459,296.656,368.489,170.542,48.066,159.298
C09871=1024.465,296.904,368.456,170.547,48.065,159.298
C09872=1024.473,297.152,368.424,170.552,48.063,159.298
C09873=1024.479,297.399,368.391,170.557,48.061,159.298
C09874=1024.485,297.648,368.359,170.562,48.059,159.299
C09875=1024.492,297.895,368.327,170.567,48.057,159.299
C09876=1024.499,298.143,368.294,170.572,48.056,159.299
C09877=1024.505,298.391,368.262,170.576,48.053,159.299
C09878=1024.512,298.639,368.229,170.581,48.052,159.300
C09879=1024.518,298.886,368.197,170.586,48.050,159.300
C09880=1024.525,299.134,368.165,170.591,48.048,159.300
C09881=1024.532,299.381,368.132,170.596,48.046,159.300
C09882=1024.539,299.629,368.099,170.601,48.045,159.301
C09883=1024.545,299.877,368.067,170.606,48.043,159.301
C09884=1024.552,300.125,368.035,170.611,48.041,159.301
C09885=1024.558,300.373,368.002,170.615,48.039,159.302
C09886=1024.566,300.621,367.969,170.621,48.037,159.302
C09887=1024.572,300.868,367.937,170.626,48.035,159.302
C09888=1024.578,301.116,367.904,170.631,48.034,159.302
C09889=1024.586,301.364,367.871,170.636,48.032,159.303
C09890=1024.592,301.611,367.839,170.641,48.030,159.303
C09891=1024.599,301.859,367.806,170.646,48.028,159.303
C09892=1024.606,302.107,367.773,170.651,48.027,159.304
C09893=1024.612,302.354,367.741,170.656,48.025,159.304
C09894=1024.619,302.602,367.708,170.660,48.023,159.304
C09895=1024.626,302.850,367.675,170.665,48.022,159.304
C09896=1024.633,303.098,367.643,170.670,48.020,159.305
C09897=1024.640,303.345,367.610,170.675,48.018,159.305
C09898=1024.646,303.593,367.577,170.680,48.016,159.305
C09899=1024.653,303.841,367.545,170.686,48.015,159.306
C09900=1024.660,304.089,367.512,170.691,48.013,159.306
C09901=1024.667,304.336,367.479,170.696,48.011,159.306
C09902=1024.674,304.585,367.446,170.701,48.010,159.307
C09903=1024.681,304.831,367.413,170.706,48.008,159.307
C09904=1024.687,305.079,367.381,170.711,48.006,159.307
C09905=1024.694,305.327,367.347,170.716,48.005,159.308
C09906=1024.701,305.575,367.315,170.721,48.003,159.308
C09907=1024.708,305.823,367.282,170.727,48.001,159.308
C09908=1024.715,306.069,367.249,170.732,47.999,159.308
C09909=1024.722,306.318,367.216,170.737,47.998,159.309
C09910=1024.728,306.542,367.186,170.741,47.997,159.309
C09911=1024.734,306.766,367.157,170.746,47.995,159.309
C09912=1024.740,306.990,367.127,170.751,47.994,159.310
C09913=1024.747,307.213,367.097,170.754,47.992,159.310
C09914=1024.753,307.438,367.068,170.759,47.990,159.310
C09915=1024.760,307.662,367.037,170.765,47.989,159.311
C09916=1024.766,307.886,367.007,170.769,47.988,159.311
C09917=1024.772,308.110,366.977,170.774,47.986,159.311
C09918=1024.780,308.358,366.945,170.779,47.985,159.312
C09919=1024.786,308.605,366.912,170.784,47.983,159.312
C09920=1024.793,308.853,366.878,170.790,47.982,159.312
C09921=1024.800,309.100,366.846,170.795,47.980,159.313
C09922=1024.808,309.348,366.812,170.800,47.979,159.313
C09923=1024.815,309.596,366.779,170.804,47.976,159.313
C09924=1024.822,309.843,366.746,170.810,47.975,159.314
C09925=1024.829,310.091,366.713,170.816,47.973,159.314
C09926=1024.836,310.339,366.679,170.821,47.972,159.314
C09927=1024.843,310.586,366.647,170.826,47.970,159.315
C09928=1024.849,310.834,366.613,170.831,47.969,159.315
C09929=1024.856,311.081,366.579,170.836,47.968,159.316
C09930=1024.863,311.329,366.545,170.841,47.967,159.316
C09931=1024.870,311.577,366.512,170.846,47.965,159.316
C09932=1024.876,311.824,366.478,170.851,47.964,159.317
C09933=1024.883,312.072,366.444,170.858,47.962,159.317
C09934=1024.890,312.319,366.411,170.863,47.961,159.318
C09935=1024.896,312.567,366.377,170.868,47.960,159.318
C09936=1024.903,312.815,366.343,170.873,47.959,159.319
C09937=1024.910,313.062,366.309,170.878,47.957,159.319
C09938=1024.917,313.310,366.275,170.883,47.956,159.320
C09939=1024.924,313.557,366.241,170.888,47.955,159.320
C09940=1024.930,313.804,366.208,170.894,47.953,159.320
C09941=1024.938,314.052,366.174,170.900,47.952,159.321
C09942=1024.944,314.300,366.139,170.905,47.951,159.321
C09943=1024.951,314.548,366.105,170.910,47.950,159.322
C09944=1024.958,314.794,366.072,170.915,47.948,159.322
C09945=1024.964,315.042,366.038,170.920,47.947,159.322
C09946=1024.971,315.290,366.004,170.927,47.946,159.323
C09947=1024.979,315.538,365.970,170.932,47.944,159.323
C09948=1024.985,315.785,365.936,170.937,47.944,159.324
C09949=1024.992,316.033,365.902,170.942,47.942,159.324
C09950=1024.999,316.280,365.868,170.947,47.941,159.325
C09951=1025.006,316.528,365.834,170.954,47.939,159.325
C09952=1025.013,316.775,365.799,170.959,47.939,159.326
C09953=1025.020,317.023,365.765,170.964,47.937,159.326
C09954=1025.027,317.270,365.732,170.969,47.936,159.327
C09955=1025.033,317.518,365.698,170.975,47.936,159.327
C09956=1025.040,317.766,365.664,170.981,47.934,159.328
C09957=1025.048,318.013,365.629,170.986,47.933,159.328
C09958=1025.054,318.261,365.595,170.991,47.931,159.329
C09959=1025.062,318.509,365.561,170.996,47.931,159.329
C09960=1025.069,318.756,365.526,171.002,47.930,159.330
C09961=1025.075,319.004,365.492,171.008,47.928,159.330
C09962=1025.083,319.251,365.458,171.013,47.927,159.331
C09963=1025.090,319.498,365.424,171.019,47.926,159.331
C09964=1025.097,319.746,365.389,171.024,47.925,159.332
C09965=1025.104,319.994,365.355,171.030,47.924,159.332
C09966=1025.111,320.241,365.321,171.035,47.923,159.333
C09967=1025.118,320.489,365.286,171.040,47.921,159.333
C09968=1025.125,320.736,365.252,171.047,47.920,159.334
C09969=1025.133,320.984,365.218,171.052,47.919,159.334
C09970=1025.138,321.210,365.187,171.057,47.918,159.335
C09971=1025.145,321.436,365.155,171.062,47.917,159.335
C09972=1025.151,321.664,365.123,171.067,47.917,159.336
C09973=1025.158,321.889,365.092,171.072,47.916,159.336
C09974=1025.165,322.116,365.061,171.077,47.914,159.336
C09975=1025.171,322.343,365.029,171.083,47.913,159.337
C09976=1025.178,322.569,364.997,171.088,47.913,159.338
C09977=1025.184,322.796,364.966,171.093,47.912,159.338
C09978=1025.192,323.044,364.931,171.099,47.911,159.339
C09979=1025.200,323.291,364.897,171.104,47.909,159.339
C09980=1025.206,323.539,364.862,171.110,47.908,159.340
C09981=1025.214,323.786,364.828,171.115,47.907,159.340
C09982=1025.220,324.034,364.793,171.121,47.907,159.341
C09983=1025.228,324.281,364.759,171.127,47.905,159.341
C09984=1025.236,324.528,364.724,171.133,47.905,159.342
C09985=1025.242,324.776,364.689,171.138,47.904,159.342
C09986=1025.250,325.024,364.655,171.144,47.903,159.343
C09987=1025.257,325.271,364.620,171.150,47.902,159.343
C09988=1025.264,325.519,364.585,171.155,47.901,159.344
C09989=1025.272,325.766,364.550,171.161,47.900,159.345
C09990=1025.279,326.013,364.517,171.167,47.899,159.345
C09991=1025.286,326.261,364.481,171.173,47.898,159.346
C09992=1025.294,326.508,364.446,171.178,47.897,159.346
C09993=1025.301,326.756,364.411,171.184,47.896,159.347
C09994=1025.308,327.003,364.377,171.190,47.895,159.347
C09995=1025.316,327.250,364.342,171.195,47.894,159.348
C09996=1025.323,327.498,364.307,171.201,47.894,159.349
//INST
///DATE 2021/06/25 14:49
///ATTR SC,RW,RJ
////FRAME ROBOT
///GROUP1 RB1
NOP
MOVL C00000 V=800.0 PL=0
MOVL C00001 V=800.0 PL=0
MOVL C00002 V=800.0 PL=0
MOVL C00003 V=800.0 PL=0
MOVL C00004 V=800.0 PL=0
MOVL C00005 V=800.0 PL=0
MOVL C00006 V=800.0 PL=0
MOVL C00007 V=800.0 PL=0
MOVL C00008 V=800.0 PL=0
MOVL C00009 V=800.0 PL=0
MOVL C00010 V=800.0 PL=0
MOVL C00011 V=800.0 PL=0
MOVL C00012 V=800.0 PL=0
MOVL C00013 V=800.0 PL=0
MOVL C00014 V=800.0 PL=0
MOVL C00015 V=800.0 PL=0
MOVL C00016 V=800.0 PL=0
MOVL C00017 V=800.0 PL=0
MOVL C00018 V=800.0 PL=0
MOVL C00019 V=800.0 PL=0
MOVL C00020 V=800.0 PL=0
MOVL C00021 V=800.0 PL=0
MOVL C00022 V=800.0 PL=0
MOVL C00023 V=800.0 PL=0
MOVL C00024 V=800.0 PL=0
MOVL C00025 V=800.0 PL=0
MOVL C00026 V=800.0 PL=0
MOVL C00027 V=800.0 PL=0
MOVL C00028 V=800.0 PL=0
MOVL C00029 V=800.0 PL=0
MOVL C00030 V=800.0 PL=0
MOVL C00031 V=800.0 PL=0
MOVL C00032 V=800.0 PL=0
MOVL C00033 V=800.0 PL=0
MOVL C00034 V=800.0 PL=0
MOVL C00035 V=800.0 PL=0
MOVL C00036 V=800.0 PL=0
MOVL C00037 V=800.0 PL=0
MOVL C00038 V=800.0 PL=0
MOVL C00039 V=800.0 PL=0
MOVL C00040 V=800.0 PL=0
MOVL C00041 V=800.0 PL=0
MOVL C00042 V=800.0 PL=0
MOVL C00043 V=800.0 PL=0
MOVL C00044 V=800.0 PL=0
MOVL C00045 V=800.0 PL=0
MOVL C00046 V=800.0 PL=0
MOVL C00047 V=800.0 PL=0
MOVL C00048 V=800.0 PL=0
MOVL C00049 V=800.0 PL=0
MOVL C00050 V=800.0 PL=0
MOVL C00051 V=800.0 PL=0
MOVL C00052 V=800.0 PL=0
MOVL C00053 V=800.0 PL=0
MOVL C00054 V=800.0 PL=0
MOVL C00055 V=800.0 PL=0
MOVL C00056 V=800.0 PL=0
MOVL C00057 V=800.0 PL=0
MOVL C00058 V=800.0 PL=0
MOVL C00059 V=800.0 PL=0
MOVL C00060 V=800.0 PL=0
MOVL C00061 V=800.0 PL=0
MOVL C00062 V=800.0 PL=0
MOVL C00063 V=800.0 PL=0
MOVL C00064 V=800.0 PL=0
MOVL C00065 V=800.0 PL=0
MOVL C00066 V=800.0 PL=0
MOVL C00067 V=800.0 PL=0
MOVL C00068 V=800.0 PL=0
MOVL C00069 V=800.0 PL=0
MOVL C00070 V=800.0 PL=0
MOVL C00071 V=800.0 PL=0
MOVL C00072 V=800.0 PL=0
MOVL C00073 V=800.0 PL=0
MOVL C00074 V=800.0 PL=0
MOVL C00075 V=800.0 PL=0
MOVL C00076 V=800.0 PL=0
MOVL C00077 V=800.0 PL=0
MOVL C00078 V=800.0 PL=0
MOVL C00079 V=800.0 PL=0
MOVL C00080 V=800.0 PL=0
MOVL C00081 V=800.0 PL=0
MOVL C00082 V=800.0 PL=0
MOVL C00083 V=800.0 PL=0
MOVL C00084 V=800.0 PL=0
MOVL C00085 V=800.0 PL=0
MOVL C00086 V=800.0 PL=0
MOVL C00087 V=800.0 PL=0
MOVL C00088 V=800.0 PL=0
MOVL C00089 V=800.0 PL=0
MOVL C00090 V=800.0 PL=0
MOVL C00091 V=800.0 PL=0
MOVL C00092 V=800.0 PL=0
MOVL C00093 V=800.0 PL=0
MOVL C00094 V=800.0 PL=0
MOVL C00095 V=800.0 PL=0
MOVL C00096 V=800.0 PL=0
MOVL C00097 V=800.0 PL=0
MOVL C00098 V=800.0 PL=0
MOVL C00099 V=800.0 PL=0
MOVL C00100 V=800.0 PL=0
MOVL C00101 V=800.0 PL=0
MOVL C00102 V=800.0 PL=0
MOVL C00103 V=800.0 PL=0
MOVL C00104 V=800.0 PL=0
MOVL C00105 V=800.0 PL=0
MOVL C00106 V=800.0 PL=0
MOVL C00107 V=800.0 PL=0
MOVL C00108 V=800.0 PL=0
MOVL C00109 V=800.0 PL=0
MOVL C00110 V=800.0 PL=0
MOVL C00111 V=800.0 PL=0
MOVL C00112 V=800.0 PL=0
MOVL C00113 V=800.0 PL=0
MOVL C00114 V=800.0 PL=0
MOVL C00115 V=800.0 PL=0
MOVL C00116 V=800.0 PL=0
MOVL C00117 V=800.0 PL=0
MOVL C00118 V=800.0 PL=0
MOVL C00119 V=800.0 PL=0
MOVL C00120 V=800.0 PL=0
MOVL C00121 V=800.0 PL=0
MOVL C00122 V=800.0 PL=0
MOVL C00123 V=800.0 PL=0
MOVL C00124 V=800.0 PL=0
MOVL C00125 V=800.0 PL=0
MOVL C00126 V=800.0 PL=0
MOVL C00127 V=800.0 PL=0
MOVL C00128 V=800.0 PL=0
MOVL C00129 V=800.0 PL=0
MOVL C00130 V=800.0 PL=0
MOVL C00131 V=800.0 PL=0
MOVL C00132 V=800.0 PL=0
MOVL C00133 V=800.0 PL=0
MOVL C00134 V=800.0 PL=0
MOVL C00135 V=800.0 PL=0
MOVL C00136 V=800.0 PL=0
MOVL C00137 V=800.0 PL=0
MOVL C00138 V=800.0 PL=0
MOVL C00139 V=800.0 PL=0
MOVL C00140 V=800.0 PL=0
MOVL C00141 V=800.0 PL=0
MOVL C00142 V=800.0 PL=0
MOVL C00143 V=800.0 PL=0
MOVL C00144 V=800.0 PL=0
MOVL C00145 V=800.0 PL=0
MOVL C00146 V=800.0 PL=0
MOVL C00147 V=800.0 PL=0
MOVL C00148 V=800.0 PL=0
MOVL C00149 V=800.0 PL=0
MOVL C00150 V=800.0 PL=0
MOVL C00151 V=800.0 PL=0
MOVL C00152 V=800.0 PL=0
MOVL C00153 V=800.0 PL=0
MOVL C00154 V=800.0 PL=0
MOVL C00155 V=800.0 PL=0
MOVL C00156 V=800.0 PL=0
MOVL C00157 V=800.0 PL=0
MOVL C00158 V=800.0 PL=0
MOVL C00159 V=800.0 PL=0
MOVL C00160 V=800.0 PL=0
MOVL C00161 V=800.0 PL=0
MOVL C00162 V=800.0 PL=0
MOVL C00163 V=800.0 PL=0
MOVL C00164 V=800.0 PL=0
MOVL C00165 V=800.0 PL=0
MOVL C00166 V=800.0 PL=0
MOVL C00167 V=800.0 PL=0
MOVL C00168 V=800.0 PL=0
MOVL C00169 V=800.0 PL=0
MOVL C00170 V=800.0 PL=0
MOVL C00171 V=800.0 PL=0
MOVL C00172 V=800.0 PL=0
MOVL C00173 V=800.0 PL=0
MOVL C00174 V=800.0 PL=0
MOVL C00175 V=800.0 PL=0
MOVL C00176 V=800.0 PL=0
MOVL C00177 V=800.0 PL=0
MOVL C00178 V=800.0 PL=0
MOVL C00179 V=800.0 PL=0
MOVL C00180 V=800.0 PL=0
MOVL C00181 V=800.0 PL=0
MOVL C00182 V=800.0 PL=0
MOVL C00183 V=800.0 PL=0
MOVL C00184 V=800.0 PL=0
MOVL C00185 V=800.0 PL=0
MOVL C00186 V=800.0 PL=0
MOVL C00187 V=800.0 PL=0
MOVL C00188 V=800.0 PL=0
MOVL C00189 V=800.0 PL=0
MOVL C00190 V=800.0 PL=0
MOVL C00191 V=800.0 PL=0
MOVL C00192 V=800.0 PL=0
MOVL C00193 V=800.0 PL=0
MOVL C00194 V=800.0 PL=0
MOVL C00195 V=800.0 PL=0
MOVL C00196 V=800.0 PL=0
MOVL C00197 V=800.0 PL=0
MOVL C00198 V=800.0 PL=0
MOVL C00199 V=800.0 PL=0
MOVL C00200 V=800.0 PL=0
MOVL C00201 V=800.0 PL=0
MOVL C00202 V=800.0 PL=0
MOVL C00203 V=800.0 PL=0
MOVL C00204 V=800.0 PL=0
MOVL C00205 V=800.0 PL=0
MOVL C00206 V=800.0 PL=0
MOVL C00207 V=800.0 PL=0
MOVL C00208 V=800.0 PL=0
MOVL C00209 V=800.0 PL=0
MOVL C00210 V=800.0 PL=0
MOVL C00211 V=800.0 PL=0
MOVL C00212 V=800.0 PL=0
MOVL C00213 V=800.0 PL=0
MOVL C00214 V=800.0 PL=0
MOVL C00215 V=800.0 PL=0
MOVL C00216 V=800.0 PL=0
MOVL C00217 V=800.0 PL=0
MOVL C00218 V=800.0 PL=0
MOVL C00219 V=800.0 PL=0
MOVL C00220 V=800.0 PL=0
MOVL C00221 V=800.0 PL=0
MOVL C00222 V=800.0 PL=0
MOVL C00223 V=800.0 PL=0
MOVL C00224 V=800.0 PL=0
MOVL C00225 V=800.0 PL=0
MOVL C00226 V=800.0 PL=0
MOVL C00227 V=800.0 PL=0
MOVL C00228 V=800.0 PL=0
MOVL C00229 V=800.0 PL=0
MOVL C00230 V=800.0 PL=0
MOVL C00231 V=800.0 PL=0
MOVL C00232 V=800.0 PL=0
MOVL C00233 V=800.0 PL=0
MOVL C00234 V=800.0 PL=0
MOVL C00235 V=800.0 PL=0
MOVL C00236 V=800.0 PL=0
MOVL C00237 V=800.0 PL=0
MOVL C00238 V=800.0 PL=0
MOVL C00239 V=800.0 PL=0
MOVL C00240 V=800.0 PL=0
MOVL C00241 V=800.0 PL=0
MOVL C00242 V=800.0 PL=0
MOVL C00243 V=800.0 PL=0
MOVL C00244 V=800.0 PL=0
MOVL C00245 V=800.0 PL=0
MOVL C00246 V=800.0 PL=0
MOVL C00247 V=800.0 PL=0
MOVL C00248 V=800.0 PL=0
MOVL C00249 V=800.0 PL=0
MOVL C00250 V=800.0 PL=0
MOVL C00251 V=800.0 PL=0
MOVL C00252 V=800.0 PL=0
MOVL C00253 V=800.0 PL=0
MOVL C00254 V=800.0 PL=0
MOVL C00255 V=800.0 PL=0
MOVL C00256 V=800.0 PL=0
MOVL C00257 V=800.0 PL=0
MOVL C00258 V=800.0 PL=0
MOVL C00259 V=800.0 PL=0
MOVL C00260 V=800.0 PL=0
MOVL C00261 V=800.0 PL=0
MOVL C00262 V=800.0 PL=0
MOVL C00263 V=800.0 PL=0
MOVL C00264 V=800.0 PL=0
MOVL C00265 V=800.0 PL=0
MOVL C00266 V=800.0 PL=0
MOVL C00267 V=800.0 PL=0
MOVL C00268 V=800.0 PL=0
MOVL C00269 V=800.0 PL=0
MOVL C00270 V=800.0 PL=0
MOVL C00271 V=800.0 PL=0
MOVL C00272 V=800.0 PL=0
MOVL C00273 V=800.0 PL=0
MOVL C00274 V=800.0 PL=0
MOVL C00275 V=800.0 PL=0
MOVL C00276 V=800.0 PL=0
MOVL C00277 V=800.0 PL=0
MOVL C00278 V=800.0 PL=0
MOVL C00279 V=800.0 PL=0
MOVL C00280 V=800.0 PL=0
MOVL C00281 V=800.0 PL=0
MOVL C00282 V=800.0 PL=0
MOVL C00283 V=800.0 PL=0
MOVL C00284 V=800.0 PL=0
MOVL C00285 V=800.0 PL=0
MOVL C00286 V=800.0 PL=0
MOVL C00287 V=800.0 PL=0
MOVL C00288 V=800.0 PL=0
MOVL C00289 V=800.0 PL=0
MOVL C00290 V=800.0 PL=0
MOVL C00291 V=800.0 PL=0
MOVL C00292 V=800.0 PL=0
MOVL C00293 V=800.0 PL=0
MOVL C00294 V=800.0 PL=0
MOVL C00295 V=800.0 PL=0
MOVL C00296 V=800.0 PL=0
MOVL C00297 V=800.0 PL=0
MOVL C00298 V=800.0 PL=0
MOVL C00299 V=800.0 PL=0
MOVL C00300 V=800.0 PL=0
MOVL C00301 V=800.0 PL=0
MOVL C00302 V=800.0 PL=0
MOVL C00303 V=800.0 PL=0
MOVL C00304 V=800.0 PL=0
MOVL C00305 V=800.0 PL=0
MOVL C00306 V=800.0 PL=0
MOVL C00307 V=800.0 PL=0
MOVL C00308 V=800.0 PL=0
MOVL C00309 V=800.0 PL=0
MOVL C00310 V=800.0 PL=0
MOVL C00311 V=800.0 PL=0
MOVL C00312 V=800.0 PL=0
MOVL C00313 V=800.0 PL=0
MOVL C00314 V=800.0 PL=0
MOVL C00315 V=800.0 PL=0
MOVL C00316 V=800.0 PL=0
MOVL C00317 V=800.0 PL=0
MOVL C00318 V=800.0 PL=0
MOVL C00319 V=800.0 PL=0
MOVL C00320 V=800.0 PL=0
MOVL C00321 V=800.0 PL=0
MOVL C00322 V=800.0 PL=0
MOVL C00323 V=800.0 PL=0
MOVL C00324 V=800.0 PL=0
MOVL C00325 V=800.0 PL=0
MOVL C00326 V=800.0 PL=0
MOVL C00327 V=800.0 PL=0
MOVL C00328 V=800.0 PL=0
MOVL C00329 V=800.0 PL=0
MOVL C00330 V=800.0 PL=0
MOVL C00331 V=800.0 PL=0
MOVL C00332 V=800.0 PL=0
MOVL C00333 V=800.0 PL=0
MOVL C00334 V=800.0 PL=0
MOVL C00335 V=800.0 PL=0
MOVL C00336 V=800.0 PL=0
MOVL C00337 V=800.0 PL=0
MOVL C00338 V=800.0 PL=0
MOVL C00339 V=800.0 PL=0
MOVL C00340 V=800.0 PL=0
MOVL C00341 V=800.0 PL=0
MOVL C00342 V=800.0 PL=0
MOVL C00343 V=800.0 PL=0
MOVL C00344 V=800.0 PL=0
MOVL C00345 V=800.0 PL=0
MOVL C00346 V=800.0 PL=0
MOVL C00347 V=800.0 PL=0
MOVL C00348 V=800.0 PL=0
MOVL C00349 V=800.0 PL=0
MOVL C00350 V=800.0 PL=0
MOVL C00351 V=800.0 PL=0
MOVL C00352 V=800.0 PL=0
MOVL C00353 V=800.0 PL=0
MOVL C00354 V=800.0 PL=0
MOVL C00355 V=800.0 PL=0
MOVL C00356 V=800.0 PL=0
MOVL C00357 V=800.0 PL=0
MOVL C00358 V=800.0 PL=0
MOVL C00359 V=800.0 PL=0
MOVL C00360 V=800.0 PL=0
MOVL C00361 V=800.0 PL=0
MOVL C00362 V=800.0 PL=0
MOVL C00363 V=800.0 PL=0
MOVL C00364 V=800.0 PL=0
MOVL C00365 V=800.0 PL=0
MOVL C00366 V=800.0 PL=0
MOVL C00367 V=800.0 PL=0
MOVL C00368 V=800.0 PL=0
MOVL C00369 V=800.0 PL=0
MOVL C00370 V=800.0 PL=0
MOVL C00371 V=800.0 PL=0
MOVL C00372 V=800.0 PL=0
MOVL C00373 V=800.0 PL=0
MOVL C00374 V=800.0 PL=0
MOVL C00375 V=800.0 PL=0
MOVL C00376 V=800.0 PL=0
MOVL C00377 V=800.0 PL=0
MOVL C00378 V=800.0 PL=0
MOVL C00379 V=800.0 PL=0
MOVL C00380 V=800.0 PL=0
MOVL C00381 V=800.0 PL=0
MOVL C00382 V=800.0 PL=0
MOVL C00383 V=800.0 PL=0
MOVL C00384 V=800.0 PL=0
MOVL C00385 V=800.0 PL=0
MOVL C00386 V=800.0 PL=0
MOVL C00387 V=800.0 PL=0
MOVL C00388 V=800.0 PL=0
MOVL C00389 V=800.0 PL=0
MOVL C00390 V=800.0 PL=0
MOVL C00391 V=800.0 PL=0
MOVL C00392 V=800.0 PL=0
MOVL C00393 V=800.0 PL=0
MOVL C00394 V=800.0 PL=0
MOVL C00395 V=800.0 PL=0
MOVL C00396 V=800.0 PL=0
MOVL C00397 V=800.0 PL=0
MOVL C00398 V=800.0 PL=0
MOVL C00399 V=800.0 PL=0
MOVL C00400 V=800.0 PL=0
MOVL C00401 V=800.0 PL=0
MOVL C00402 V=800.0 PL=0
MOVL C00403 V=800.0 PL=0
MOVL C00404 V=800.0 PL=0
MOVL C00405 V=800.0 PL=0
MOVL C00406 V=800.0 PL=0
MOVL C00407 V=800.0 PL=0
MOVL C00408 V=800.0 PL=0
MOVL C00409 V=800.0 PL=0
MOVL C00410 V=800.0 PL=0
MOVL C00411 V=800.0 PL=0
MOVL C00412 V=800.0 PL=0
MOVL C00413 V=800.0 PL=0
MOVL C00414 V=800.0 PL=0
MOVL C00415 V=800.0 PL=0
MOVL C00416 V=800.0 PL=0
MOVL C00417 V=800.0 PL=0
MOVL C00418 V=800.0 PL=0
MOVL C00419 V=800.0 PL=0
MOVL C00420 V=800.0 PL=0
MOVL C00421 V=800.0 PL=0
MOVL C00422 V=800.0 PL=0
MOVL C00423 V=800.0 PL=0
MOVL C00424 V=800.0 PL=0
MOVL C00425 V=800.0 PL=0
MOVL C00426 V=800.0 PL=0
MOVL C00427 V=800.0 PL=0
MOVL C00428 V=800.0 PL=0
MOVL C00429 V=800.0 PL=0
MOVL C00430 V=800.0 PL=0
MOVL C00431 V=800.0 PL=0
MOVL C00432 V=800.0 PL=0
MOVL C00433 V=800.0 PL=0
MOVL C00434 V=800.0 PL=0
MOVL C00435 V=800.0 PL=0
MOVL C00436 V=800.0 PL=0
MOVL C00437 V=800.0 PL=0
MOVL C00438 V=800.0 PL=0
MOVL C00439 V=800.0 PL=0
MOVL C00440 V=800.0 PL=0
MOVL C00441 V=800.0 PL=0
MOVL C00442 V=800.0 PL=0
MOVL C00443 V=800.0 PL=0
MOVL C00444 V=800.0 PL=0
MOVL C00445 V=800.0 PL=0
MOVL C00446 V=800.0 PL=0
MOVL C00447 V=800.0 PL=0
MOVL C00448 V=800.0 PL=0
MOVL C00449 V=800.0 PL=0
MOVL C00450 V=800.0 PL=0
MOVL C00451 V=800.0 PL=0
MOVL C00452 V=800.0 PL=0
MOVL C00453 V=800.0 PL=0
MOVL C00454 V=800.0 PL=0
MOVL C00455 V=800.0 PL=0
MOVL C00456 V=800.0 PL=0
MOVL C00457 V=800.0 PL=0
MOVL C00458 V=800.0 PL=0
MOVL C00459 V=800.0 PL=0
MOVL C00460 V=800.0 PL=0
MOVL C00461 V=800.0 PL=0
MOVL C00462 V=800.0 PL=0
MOVL C00463 V=800.0 PL=0
MOVL C00464 V=800.0 PL=0
MOVL C00465 V=800.0 PL=0
MOVL C00466 V=800.0 PL=0
MOVL C00467 V=800.0 PL=0
MOVL C00468 V=800.0 PL=0
MOVL C00469 V=800.0 PL=0
MOVL C00470 V=800.0 PL=0
MOVL C00471 V=800.0 PL=0
MOVL C00472 V=800.0 PL=0
MOVL C00473 V=800.0 PL=0
MOVL C00474 V=800.0 PL=0
MOVL C00475 V=800.0 PL=0
MOVL C00476 V=800.0 PL=0
MOVL C00477 V=800.0 PL=0
MOVL C00478 V=800.0 PL=0
MOVL C00479 V=800.0 PL=0
MOVL C00480 V=800.0 PL=0
MOVL C00481 V=800.0 PL=0
MOVL C00482 V=800.0 PL=0
MOVL C00483 V=800.0 PL=0
MOVL C00484 V=800.0 PL=0
MOVL C00485 V=800.0 PL=0
MOVL C00486 V=800.0 PL=0
MOVL C00487 V=800.0 PL=0
MOVL C00488 V=800.0 PL=0
MOVL C00489 V=800.0 PL=0
MOVL C00490 V=800.0 PL=0
MOVL C00491 V=800.0 PL=0
MOVL C00492 V=800.0 PL=0
MOVL C00493 V=800.0 PL=0
MOVL C00494 V=800.0 PL=0
MOVL C00495 V=800.0 PL=0
MOVL C00496 V=800.0 PL=0
MOVL C00497 V=800.0 PL=0
MOVL C00498 V=800.0 PL=0
MOVL C00499 V=800.0 PL=0
MOVL C00500 V=800.0 PL=0
MOVL C00501 V=800.0 PL=0
MOVL C00502 V=800.0 PL=0
MOVL C00503 V=800.0 PL=0
MOVL C00504 V=800.0 PL=0
MOVL C00505 V=800.0 PL=0
MOVL C00506 V=800.0 PL=0
MOVL C00507 V=800.0 PL=0
MOVL C00508 V=800.0 PL=0
MOVL C00509 V=800.0 PL=0
MOVL C00510 V=800.0 PL=0
MOVL C00511 V=800.0 PL=0
MOVL C00512 V=800.0 PL=0
MOVL C00513 V=800.0 PL=0
MOVL C00514 V=800.0 PL=0
MOVL C00515 V=800.0 PL=0
MOVL C00516 V=800.0 PL=0
MOVL C00517 V=800.0 PL=0
MOVL C00518 V=800.0 PL=0
MOVL C00519 V=800.0 PL=0
MOVL C00520 V=800.0 PL=0
MOVL C00521 V=800.0 PL=0
MOVL C00522 V=800.0 PL=0
MOVL C00523 V=800.0 PL=0
MOVL C00524 V=800.0 PL=0
MOVL C00525 V=800.0 PL=0
MOVL C00526 V=800.0 PL=0
MOVL C00527 V=800.0 PL=0
MOVL C00528 V=800.0 PL=0
MOVL C00529 V=800.0 PL=0
MOVL C00530 V=800.0 PL=0
MOVL C00531 V=800.0 PL=0
MOVL C00532 V=800.0 PL=0
MOVL C00533 V=800.0 PL=0
MOVL C00534 V=800.0 PL=0
MOVL C00535 V=800.0 PL=0
MOVL C00536 V=800.0 PL=0
MOVL C00537 V=800.0 PL=0
MOVL C00538 V=800.0 PL=0
MOVL C00539 V=800.0 PL=0
MOVL C00540 V=800.0 PL=0
MOVL C00541 V=800.0 PL=0
MOVL C00542 V=800.0 PL=0
MOVL C00543 V=800.0 PL=0
MOVL C00544 V=800.0 PL=0
MOVL C00545 V=800.0 PL=0
MOVL C00546 V=800.0 PL=0
MOVL C00547 V=800.0 PL=0
MOVL C00548 V=800.0 PL=0
MOVL C00549 V=800.0 PL=0
MOVL C00550 V=800.0 PL=0
MOVL C00551 V=800.0 PL=0
MOVL C00552 V=800.0 PL=0
MOVL C00553 V=800.0 PL=0
MOVL C00554 V=800.0 PL=0
MOVL C00555 V=800.0 PL=0
MOVL C00556 V=800.0 PL=0
MOVL C00557 V=800.0 PL=0
MOVL C00558 V=800.0 PL=0
MOVL C00559 V=800.0 PL=0
MOVL C00560 V=800.0 PL=0
MOVL C00561 V=800.0 PL=0
MOVL C00562 V=800.0 PL=0
MOVL C00563 V=800.0 PL=0
MOVL C00564 V=800.0 PL=0
MOVL C00565 V=800.0 PL=0
MOVL C00566 V=800.0 PL=0
MOVL C00567 V=800.0 PL=0
MOVL C00568 V=800.0 PL=0
MOVL C00569 V=800.0 PL=0
MOVL C00570 V=800.0 PL=0
MOVL C00571 V=800.0 PL=0
MOVL C00572 V=800.0 PL=0
MOVL C00573 V=800.0 PL=0
MOVL C00574 V=800.0 PL=0
MOVL C00575 V=800.0 PL=0
MOVL C00576 V=800.0 PL=0
MOVL C00577 V=800.0 PL=0
MOVL C00578 V=800.0 PL=0
MOVL C00579 V=800.0 PL=0
MOVL C00580 V=800.0 PL=0
MOVL C00581 V=800.0 PL=0
MOVL C00582 V=800.0 PL=0
MOVL C00583 V=800.0 PL=0
MOVL C00584 V=800.0 PL=0
MOVL C00585 V=800.0 PL=0
MOVL C00586 V=800.0 PL=0
MOVL C00587 V=800.0 PL=0
MOVL C00588 V=800.0 PL=0
MOVL C00589 V=800.0 PL=0
MOVL C00590 V=800.0 PL=0
MOVL C00591 V=800.0 PL=0
MOVL C00592 V=800.0 PL=0
MOVL C00593 V=800.0 PL=0
MOVL C00594 V=800.0 PL=0
MOVL C00595 V=800.0 PL=0
MOVL C00596 V=800.0 PL=0
MOVL C00597 V=800.0 PL=0
MOVL C00598 V=800.0 PL=0
MOVL C00599 V=800.0 PL=0
MOVL C00600 V=800.0 PL=0
MOVL C00601 V=800.0 PL=0
MOVL C00602 V=800.0 PL=0
MOVL C00603 V=800.0 PL=0
MOVL C00604 V=800.0 PL=0
MOVL C00605 V=800.0 PL=0
MOVL C00606 V=800.0 PL=0
MOVL C00607 V=800.0 PL=0
MOVL C00608 V=800.0 PL=0
MOVL C00609 V=800.0 PL=0
MOVL C00610 V=800.0 PL=0
MOVL C00611 V=800.0 PL=0
MOVL C00612 V=800.0 PL=0
MOVL C00613 V=800.0 PL=0
MOVL C00614 V=800.0 PL=0
MOVL C00615 V=800.0 PL=0
MOVL C00616 V=800.0 PL=0
MOVL C00617 V=800.0 PL=0
MOVL C00618 V=800.0 PL=0
MOVL C00619 V=800.0 PL=0
MOVL C00620 V=800.0 PL=0
MOVL C00621 V=800.0 PL=0
MOVL C00622 V=800.0 PL=0
MOVL C00623 V=800.0 PL=0
MOVL C00624 V=800.0 PL=0
MOVL C00625 V=800.0 PL=0
MOVL C00626 V=800.0 PL=0
MOVL C00627 V=800.0 PL=0
MOVL C00628 V=800.0 PL=0
MOVL C00629 V=800.0 PL=0
MOVL C00630 V=800.0 PL=0
MOVL C00631 V=800.0 PL=0
MOVL C00632 V=800.0 PL=0
MOVL C00633 V=800.0 PL=0
MOVL C00634 V=800.0 PL=0
MOVL C00635 V=800.0 PL=0
MOVL C00636 V=800.0 PL=0
MOVL C00637 V=800.0 PL=0
MOVL C00638 V=800.0 PL=0
MOVL C00639 V=800.0 PL=0
MOVL C00640 V=800.0 PL=0
MOVL C00641 V=800.0 PL=0
MOVL C00642 V=800.0 PL=0
MOVL C00643 V=800.0 PL=0
MOVL C00644 V=800.0 PL=0
MOVL C00645 V=800.0 PL=0
MOVL C00646 V=800.0 PL=0
MOVL C00647 V=800.0 PL=0
MOVL C00648 V=800.0 PL=0
MOVL C00649 V=800.0 PL=0
MOVL C00650 V=800.0 PL=0
MOVL C00651 V=800.0 PL=0
MOVL C00652 V=800.0 PL=0
MOVL C00653 V=800.0 PL=0
MOVL C00654 V=800.0 PL=0
MOVL C00655 V=800.0 PL=0
MOVL C00656 V=800.0 PL=0
MOVL C00657 V=800.0 PL=0
MOVL C00658 V=800.0 PL=0
MOVL C00659 V=800.0 PL=0
MOVL C00660 V=800.0 PL=0
MOVL C00661 V=800.0 PL=0
MOVL C00662 V=800.0 PL=0
MOVL C00663 V=800.0 PL=0
MOVL C00664 V=800.0 PL=0
MOVL C00665 V=800.0 PL=0
MOVL C00666 V=800.0 PL=0
MOVL C00667 V=800.0 PL=0
MOVL C00668 V=800.0 PL=0
MOVL C00669 V=800.0 PL=0
MOVL C00670 V=800.0 PL=0
MOVL C00671 V=800.0 PL=0
MOVL C00672 V=800.0 PL=0
MOVL C00673 V=800.0 PL=0
MOVL C00674 V=800.0 PL=0
MOVL C00675 V=800.0 PL=0
MOVL C00676 V=800.0 PL=0
MOVL C00677 V=800.0 PL=0
MOVL C00678 V=800.0 PL=0
MOVL C00679 V=800.0 PL=0
MOVL C00680 V=800.0 PL=0
MOVL C00681 V=800.0 PL=0
MOVL C00682 V=800.0 PL=0
MOVL C00683 V=800.0 PL=0
MOVL C00684 V=800.0 PL=0
MOVL C00685 V=800.0 PL=0
MOVL C00686 V=800.0 PL=0
MOVL C00687 V=800.0 PL=0
MOVL C00688 V=800.0 PL=0
MOVL C00689 V=800.0 PL=0
MOVL C00690 V=800.0 PL=0
MOVL C00691 V=800.0 PL=0
MOVL C00692 V=800.0 PL=0
MOVL C00693 V=800.0 PL=0
MOVL C00694 V=800.0 PL=0
MOVL C00695 V=800.0 PL=0
MOVL C00696 V=800.0 PL=0
MOVL C00697 V=800.0 PL=0
MOVL C00698 V=800.0 PL=0
MOVL C00699 V=800.0 PL=0
MOVL C00700 V=800.0 PL=0
MOVL C00701 V=800.0 PL=0
MOVL C00702 V=800.0 PL=0
MOVL C00703 V=800.0 PL=0
MOVL C00704 V=800.0 PL=0
MOVL C00705 V=800.0 PL=0
MOVL C00706 V=800.0 PL=0
MOVL C00707 V=800.0 PL=0
MOVL C00708 V=800.0 PL=0
MOVL C00709 V=800.0 PL=0
MOVL C00710 V=800.0 PL=0
MOVL C00711 V=800.0 PL=0
MOVL C00712 V=800.0 PL=0
MOVL C00713 V=800.0 PL=0
MOVL C00714 V=800.0 PL=0
MOVL C00715 V=800.0 PL=0
MOVL C00716 V=800.0 PL=0
MOVL C00717 V=800.0 PL=0
MOVL C00718 V=800.0 PL=0
MOVL C00719 V=800.0 PL=0
MOVL C00720 V=800.0 PL=0
MOVL C00721 V=800.0 PL=0
MOVL C00722 V=800.0 PL=0
MOVL C00723 V=800.0 PL=0
MOVL C00724 V=800.0 PL=0
MOVL C00725 V=800.0 PL=0
MOVL C00726 V=800.0 PL=0
MOVL C00727 V=800.0 PL=0
MOVL C00728 V=800.0 PL=0
MOVL C00729 V=800.0 PL=0
MOVL C00730 V=800.0 PL=0
MOVL C00731 V=800.0 PL=0
MOVL C00732 V=800.0 PL=0
MOVL C00733 V=800.0 PL=0
MOVL C00734 V=800.0 PL=0
MOVL C00735 V=800.0 PL=0
MOVL C00736 V=800.0 PL=0
MOVL C00737 V=800.0 PL=0
MOVL C00738 V=800.0 PL=0
MOVL C00739 V=800.0 PL=0
MOVL C00740 V=800.0 PL=0
MOVL C00741 V=800.0 PL=0
MOVL C00742 V=800.0 PL=0
MOVL C00743 V=800.0 PL=0
MOVL C00744 V=800.0 PL=0
MOVL C00745 V=800.0 PL=0
MOVL C00746 V=800.0 PL=0
MOVL C00747 V=800.0 PL=0
MOVL C00748 V=800.0 PL=0
MOVL C00749 V=800.0 PL=0
MOVL C00750 V=800.0 PL=0
MOVL C00751 V=800.0 PL=0
MOVL C00752 V=800.0 PL=0
MOVL C00753 V=800.0 PL=0
MOVL C00754 V=800.0 PL=0
MOVL C00755 V=800.0 PL=0
MOVL C00756 V=800.0 PL=0
MOVL C00757 V=800.0 PL=0
MOVL C00758 V=800.0 PL=0
MOVL C00759 V=800.0 PL=0
MOVL C00760 V=800.0 PL=0
MOVL C00761 V=800.0 PL=0
MOVL C00762 V=800.0 PL=0
MOVL C00763 V=800.0 PL=0
MOVL C00764 V=800.0 PL=0
MOVL C00765 V=800.0 PL=0
MOVL C00766 V=800.0 PL=0
MOVL C00767 V=800.0 PL=0
MOVL C00768 V=800.0 PL=0
MOVL C00769 V=800.0 PL=0
MOVL C00770 V=800.0 PL=0
MOVL C00771 V=800.0 PL=0
MOVL C00772 V=800.0 PL=0
MOVL C00773 V=800.0 PL=0
MOVL C00774 V=800.0 PL=0
MOVL C00775 V=800.0 PL=0
MOVL C00776 V=800.0 PL=0
MOVL C00777 V=800.0 PL=0
MOVL C00778 V=800.0 PL=0
MOVL C00779 V=800.0 PL=0
MOVL C00780 V=800.0 PL=0
MOVL C00781 V=800.0 PL=0
MOVL C00782 V=800.0 PL=0
MOVL C00783 V=800.0 PL=0
MOVL C00784 V=800.0 PL=0
MOVL C00785 V=800.0 PL=0
MOVL C00786 V=800.0 PL=0
MOVL C00787 V=800.0 PL=0
MOVL C00788 V=800.0 PL=0
MOVL C00789 V=800.0 PL=0
MOVL C00790 V=800.0 PL=0
MOVL C00791 V=800.0 PL=0
MOVL C00792 V=800.0 PL=0
MOVL C00793 V=800.0 PL=0
MOVL C00794 V=800.0 PL=0
MOVL C00795 V=800.0 PL=0
MOVL C00796 V=800.0 PL=0
MOVL C00797 V=800.0 PL=0
MOVL C00798 V=800.0 PL=0
MOVL C00799 V=800.0 PL=0
MOVL C00800 V=800.0 PL=0
MOVL C00801 V=800.0 PL=0
MOVL C00802 V=800.0 PL=0
MOVL C00803 V=800.0 PL=0
MOVL C00804 V=800.0 PL=0
MOVL C00805 V=800.0 PL=0
MOVL C00806 V=800.0 PL=0
MOVL C00807 V=800.0 PL=0
MOVL C00808 V=800.0 PL=0
MOVL C00809 V=800.0 PL=0
MOVL C00810 V=800.0 PL=0
MOVL C00811 V=800.0 PL=0
MOVL C00812 V=800.0 PL=0
MOVL C00813 V=800.0 PL=0
MOVL C00814 V=800.0 PL=0
MOVL C00815 V=800.0 PL=0
MOVL C00816 V=800.0 PL=0
MOVL C00817 V=800.0 PL=0
MOVL C00818 V=800.0 PL=0
MOVL C00819 V=800.0 PL=0
MOVL C00820 V=800.0 PL=0
MOVL C00821 V=800.0 PL=0
MOVL C00822 V=800.0 PL=0
MOVL C00823 V=800.0 PL=0
MOVL C00824 V=800.0 PL=0
MOVL C00825 V=800.0 PL=0
MOVL C00826 V=800.0 PL=0
MOVL C00827 V=800.0 PL=0
MOVL C00828 V=800.0 PL=0
MOVL C00829 V=800.0 PL=0
MOVL C00830 V=800.0 PL=0
MOVL C00831 V=800.0 PL=0
MOVL C00832 V=800.0 PL=0
MOVL C00833 V=800.0 PL=0
MOVL C00834 V=800.0 PL=0
MOVL C00835 V=800.0 PL=0
MOVL C00836 V=800.0 PL=0
MOVL C00837 V=800.0 PL=0
MOVL C00838 V=800.0 PL=0
MOVL C00839 V=800.0 PL=0
MOVL C00840 V=800.0 PL=0
MOVL C00841 V=800.0 PL=0
MOVL C00842 V=800.0 PL=0
MOVL C00843 V=800.0 PL=0
MOVL C00844 V=800.0 PL=0
MOVL C00845 V=800.0 PL=0
MOVL C00846 V=800.0 PL=0
MOVL C00847 V=800.0 PL=0
MOVL C00848 V=800.0 PL=0
MOVL C00849 V=800.0 PL=0
MOVL C00850 V=800.0 PL=0
MOVL C00851 V=800.0 PL=0
MOVL C00852 V=800.0 PL=0
MOVL C00853 V=800.0 PL=0
MOVL C00854 V=800.0 PL=0
MOVL C00855 V=800.0 PL=0
MOVL C00856 V=800.0 PL=0
MOVL C00857 V=800.0 PL=0
MOVL C00858 V=800.0 PL=0
MOVL C00859 V=800.0 PL=0
MOVL C00860 V=800.0 PL=0
MOVL C00861 V=800.0 PL=0
MOVL C00862 V=800.0 PL=0
MOVL C00863 V=800.0 PL=0
MOVL C00864 V=800.0 PL=0
MOVL C00865 V=800.0 PL=0
MOVL C00866 V=800.0 PL=0
MOVL C00867 V=800.0 PL=0
MOVL C00868 V=800.0 PL=0
MOVL C00869 V=800.0 PL=0
MOVL C00870 V=800.0 PL=0
MOVL C00871 V=800.0 PL=0
MOVL C00872 V=800.0 PL=0
MOVL C00873 V=800.0 PL=0
MOVL C00874 V=800.0 PL=0
MOVL C00875 V=800.0 PL=0
MOVL C00876 V=800.0 PL=0
MOVL C00877 V=800.0 PL=0
MOVL C00878 V=800.0 PL=0
MOVL C00879 V=800.0 PL=0
MOVL C00880 V=800.0 PL=0
MOVL C00881 V=800.0 PL=0
MOVL C00882 V=800.0 PL=0
MOVL C00883 V=800.0 PL=0
MOVL C00884 V=800.0 PL=0
MOVL C00885 V=800.0 PL=0
MOVL C00886 V=800.0 PL=0
MOVL C00887 V=800.0 PL=0
MOVL C00888 V=800.0 PL=0
MOVL C00889 V=800.0 PL=0
MOVL C00890 V=800.0 PL=0
MOVL C00891 V=800.0 PL=0
MOVL C00892 V=800.0 PL=0
MOVL C00893 V=800.0 PL=0
MOVL C00894 V=800.0 PL=0
MOVL C00895 V=800.0 PL=0
MOVL C00896 V=800.0 PL=0
MOVL C00897 V=800.0 PL=0
MOVL C00898 V=800.0 PL=0
MOVL C00899 V=800.0 PL=0
MOVL C00900 V=800.0 PL=0
MOVL C00901 V=800.0 PL=0
MOVL C00902 V=800.0 PL=0
MOVL C00903 V=800.0 PL=0
MOVL C00904 V=800.0 PL=0
MOVL C00905 V=800.0 PL=0
MOVL C00906 V=800.0 PL=0
MOVL C00907 V=800.0 PL=0
MOVL C00908 V=800.0 PL=0
MOVL C00909 V=800.0 PL=0
MOVL C00910 V=800.0 PL=0
MOVL C00911 V=800.0 PL=0
MOVL C00912 V=800.0 PL=0
MOVL C00913 V=800.0 PL=0
MOVL C00914 V=800.0 PL=0
MOVL C00915 V=800.0 PL=0
MOVL C00916 V=800.0 PL=0
MOVL C00917 V=800.0 PL=0
MOVL C00918 V=800.0 PL=0
MOVL C00919 V=800.0 PL=0
MOVL C00920 V=800.0 PL=0
MOVL C00921 V=800.0 PL=0
MOVL C00922 V=800.0 PL=0
MOVL C00923 V=800.0 PL=0
MOVL C00924 V=800.0 PL=0
MOVL C00925 V=800.0 PL=0
MOVL C00926 V=800.0 PL=0
MOVL C00927 V=800.0 PL=0
MOVL C00928 V=800.0 PL=0
MOVL C00929 V=800.0 PL=0
MOVL C00930 V=800.0 PL=0
MOVL C00931 V=800.0 PL=0
MOVL C00932 V=800.0 PL=0
MOVL C00933 V=800.0 PL=0
MOVL C00934 V=800.0 PL=0
MOVL C00935 V=800.0 PL=0
MOVL C00936 V=800.0 PL=0
MOVL C00937 V=800.0 PL=0
MOVL C00938 V=800.0 PL=0
MOVL C00939 V=800.0 PL=0
MOVL C00940 V=800.0 PL=0
MOVL C00941 V=800.0 PL=0
MOVL C00942 V=800.0 PL=0
MOVL C00943 V=800.0 PL=0
MOVL C00944 V=800.0 PL=0
MOVL C00945 V=800.0 PL=0
MOVL C00946 V=800.0 PL=0
MOVL C00947 V=800.0 PL=0
MOVL C00948 V=800.0 PL=0
MOVL C00949 V=800.0 PL=0
MOVL C00950 V=800.0 PL=0
MOVL C00951 V=800.0 PL=0
MOVL C00952 V=800.0 PL=0
MOVL C00953 V=800.0 PL=0
MOVL C00954 V=800.0 PL=0
MOVL C00955 V=800.0 PL=0
MOVL C00956 V=800.0 PL=0
MOVL C00957 V=800.0 PL=0
MOVL C00958 V=800.0 PL=0
MOVL C00959 V=800.0 PL=0
MOVL C00960 V=800.0 PL=0
MOVL C00961 V=800.0 PL=0
MOVL C00962 V=800.0 PL=0
MOVL C00963 V=800.0 PL=0
MOVL C00964 V=800.0 PL=0
MOVL C00965 V=800.0 PL=0
MOVL C00966 V=800.0 PL=0
MOVL C00967 V=800.0 PL=0
MOVL C00968 V=800.0 PL=0
MOVL C00969 V=800.0 PL=0
MOVL C00970 V=800.0 PL=0
MOVL C00971 V=800.0 PL=0
MOVL C00972 V=800.0 PL=0
MOVL C00973 V=800.0 PL=0
MOVL C00974 V=800.0 PL=0
MOVL C00975 V=800.0 PL=0
MOVL C00976 V=800.0 PL=0
MOVL C00977 V=800.0 PL=0
MOVL C00978 V=800.0 PL=0
MOVL C00979 V=800.0 PL=0
MOVL C00980 V=800.0 PL=0
MOVL C00981 V=800.0 PL=0
MOVL C00982 V=800.0 PL=0
MOVL C00983 V=800.0 PL=0
MOVL C00984 V=800.0 PL=0
MOVL C00985 V=800.0 PL=0
MOVL C00986 V=800.0 PL=0
MOVL C00987 V=800.0 PL=0
MOVL C00988 V=800.0 PL=0
MOVL C00989 V=800.0 PL=0
MOVL C00990 V=800.0 PL=0
MOVL C00991 V=800.0 PL=0
MOVL C00992 V=800.0 PL=0
MOVL C00993 V=800.0 PL=0
MOVL C00994 V=800.0 PL=0
MOVL C00995 V=800.0 PL=0
MOVL C00996 V=800.0 PL=0
MOVL C00997 V=800.0 PL=0
MOVL C00998 V=800.0 PL=0
MOVL C00999 V=800.0 PL=0
MOVL C01000 V=800.0 PL=0
MOVL C01001 V=800.0 PL=0
MOVL C01002 V=800.0 PL=0
MOVL C01003 V=800.0 PL=0
MOVL C01004 V=800.0 PL=0
MOVL C01005 V=800.0 PL=0
MOVL C01006 V=800.0 PL=0
MOVL C01007 V=800.0 PL=0
MOVL C01008 V=800.0 PL=0
MOVL C01009 V=800.0 PL=0
MOVL C01010 V=800.0 PL=0
MOVL C01011 V=800.0 PL=0
MOVL C01012 V=800.0 PL=0
MOVL C01013 V=800.0 PL=0
MOVL C01014 V=800.0 PL=0
MOVL C01015 V=800.0 PL=0
MOVL C01016 V=800.0 PL=0
MOVL C01017 V=800.0 PL=0
MOVL C01018 V=800.0 PL=0
MOVL C01019 V=800.0 PL=0
MOVL C01020 V=800.0 PL=0
MOVL C01021 V=800.0 PL=0
MOVL C01022 V=800.0 PL=0
MOVL C01023 V=800.0 PL=0
MOVL C01024 V=800.0 PL=0
MOVL C01025 V=800.0 PL=0
MOVL C01026 V=800.0 PL=0
MOVL C01027 V=800.0 PL=0
MOVL C01028 V=800.0 PL=0
MOVL C01029 V=800.0 PL=0
MOVL C01030 V=800.0 PL=0
MOVL C01031 V=800.0 PL=0
MOVL C01032 V=800.0 PL=0
MOVL C01033 V=800.0 PL=0
MOVL C01034 V=800.0 PL=0
MOVL C01035 V=800.0 PL=0
MOVL C01036 V=800.0 PL=0
MOVL C01037 V=800.0 PL=0
MOVL C01038 V=800.0 PL=0
MOVL C01039 V=800.0 PL=0
MOVL C01040 V=800.0 PL=0
MOVL C01041 V=800.0 PL=0
MOVL C01042 V=800.0 PL=0
MOVL C01043 V=800.0 PL=0
MOVL C01044 V=800.0 PL=0
MOVL C01045 V=800.0 PL=0
MOVL C01046 V=800.0 PL=0
MOVL C01047 V=800.0 PL=0
MOVL C01048 V=800.0 PL=0
MOVL C01049 V=800.0 PL=0
MOVL C01050 V=800.0 PL=0
MOVL C01051 V=800.0 PL=0
MOVL C01052 V=800.0 PL=0
MOVL C01053 V=800.0 PL=0
MOVL C01054 V=800.0 PL=0
MOVL C01055 V=800.0 PL=0
MOVL C01056 V=800.0 PL=0
MOVL C01057 V=800.0 PL=0
MOVL C01058 V=800.0 PL=0
MOVL C01059 V=800.0 PL=0
MOVL C01060 V=800.0 PL=0
MOVL C01061 V=800.0 PL=0
MOVL C01062 V=800.0 PL=0
MOVL C01063 V=800.0 PL=0
MOVL C01064 V=800.0 PL=0
MOVL C01065 V=800.0 PL=0
MOVL C01066 V=800.0 PL=0
MOVL C01067 V=800.0 PL=0
MOVL C01068 V=800.0 PL=0
MOVL C01069 V=800.0 PL=0
MOVL C01070 V=800.0 PL=0
MOVL C01071 V=800.0 PL=0
MOVL C01072 V=800.0 PL=0
MOVL C01073 V=800.0 PL=0
MOVL C01074 V=800.0 PL=0
MOVL C01075 V=800.0 PL=0
MOVL C01076 V=800.0 PL=0
MOVL C01077 V=800.0 PL=0
MOVL C01078 V=800.0 PL=0
MOVL C01079 V=800.0 PL=0
MOVL C01080 V=800.0 PL=0
MOVL C01081 V=800.0 PL=0
MOVL C01082 V=800.0 PL=0
MOVL C01083 V=800.0 PL=0
MOVL C01084 V=800.0 PL=0
MOVL C01085 V=800.0 PL=0
MOVL C01086 V=800.0 PL=0
MOVL C01087 V=800.0 PL=0
MOVL C01088 V=800.0 PL=0
MOVL C01089 V=800.0 PL=0
MOVL C01090 V=800.0 PL=0
MOVL C01091 V=800.0 PL=0
MOVL C01092 V=800.0 PL=0
MOVL C01093 V=800.0 PL=0
MOVL C01094 V=800.0 PL=0
MOVL C01095 V=800.0 PL=0
MOVL C01096 V=800.0 PL=0
MOVL C01097 V=800.0 PL=0
MOVL C01098 V=800.0 PL=0
MOVL C01099 V=800.0 PL=0
MOVL C01100 V=800.0 PL=0
MOVL C01101 V=800.0 PL=0
MOVL C01102 V=800.0 PL=0
MOVL C01103 V=800.0 PL=0
MOVL C01104 V=800.0 PL=0
MOVL C01105 V=800.0 PL=0
MOVL C01106 V=800.0 PL=0
MOVL C01107 V=800.0 PL=0
MOVL C01108 V=800.0 PL=0
MOVL C01109 V=800.0 PL=0
MOVL C01110 V=800.0 PL=0
MOVL C01111 V=800.0 PL=0
MOVL C01112 V=800.0 PL=0
MOVL C01113 V=800.0 PL=0
MOVL C01114 V=800.0 PL=0
MOVL C01115 V=800.0 PL=0
MOVL C01116 V=800.0 PL=0
MOVL C01117 V=800.0 PL=0
MOVL C01118 V=800.0 PL=0
MOVL C01119 V=800.0 PL=0
MOVL C01120 V=800.0 PL=0
MOVL C01121 V=800.0 PL=0
MOVL C01122 V=800.0 PL=0
MOVL C01123 V=800.0 PL=0
MOVL C01124 V=800.0 PL=0
MOVL C01125 V=800.0 PL=0
MOVL C01126 V=800.0 PL=0
MOVL C01127 V=800.0 PL=0
MOVL C01128 V=800.0 PL=0
MOVL C01129 V=800.0 PL=0
MOVL C01130 V=800.0 PL=0
MOVL C01131 V=800.0 PL=0
MOVL C01132 V=800.0 PL=0
MOVL C01133 V=800.0 PL=0
MOVL C01134 V=800.0 PL=0
MOVL C01135 V=800.0 PL=0
MOVL C01136 V=800.0 PL=0
MOVL C01137 V=800.0 PL=0
MOVL C01138 V=800.0 PL=0
MOVL C01139 V=800.0 PL=0
MOVL C01140 V=800.0 PL=0
MOVL C01141 V=800.0 PL=0
MOVL C01142 V=800.0 PL=0
MOVL C01143 V=800.0 PL=0
MOVL C01144 V=800.0 PL=0
MOVL C01145 V=800.0 PL=0
MOVL C01146 V=800.0 PL=0
MOVL C01147 V=800.0 PL=0
MOVL C01148 V=800.0 PL=0
MOVL C01149 V=800.0 PL=0
MOVL C01150 V=800.0 PL=0
MOVL C01151 V=800.0 PL=0
MOVL C01152 V=800.0 PL=0
MOVL C01153 V=800.0 PL=0
MOVL C01154 V=800.0 PL=0
MOVL C01155 V=800.0 PL=0
MOVL C01156 V=800.0 PL=0
MOVL C01157 V=800.0 PL=0
MOVL C01158 V=800.0 PL=0
MOVL C01159 V=800.0 PL=0
MOVL C01160 V=800.0 PL=0
MOVL C01161 V=800.0 PL=0
MOVL C01162 V=800.0 PL=0
MOVL C01163 V=800.0 PL=0
MOVL C01164 V=800.0 PL=0
MOVL C01165 V=800.0 PL=0
MOVL C01166 V=800.0 PL=0
MOVL C01167 V=800.0 PL=0
MOVL C01168 V=800.0 PL=0
MOVL C01169 V=800.0 PL=0
MOVL C01170 V=800.0 PL=0
MOVL C01171 V=800.0 PL=0
MOVL C01172 V=800.0 PL=0
MOVL C01173 V=800.0 PL=0
MOVL C01174 V=800.0 PL=0
MOVL C01175 V=800.0 PL=0
MOVL C01176 V=800.0 PL=0
MOVL C01177 V=800.0 PL=0
MOVL C01178 V=800.0 PL=0
MOVL C01179 V=800.0 PL=0
MOVL C01180 V=800.0 PL=0
MOVL C01181 V=800.0 PL=0
MOVL C01182 V=800.0 PL=0
MOVL C01183 V=800.0 PL=0
MOVL C01184 V=800.0 PL=0
MOVL C01185 V=800.0 PL=0
MOVL C01186 V=800.0 PL=0
MOVL C01187 V=800.0 PL=0
MOVL C01188 V=800.0 PL=0
MOVL C01189 V=800.0 PL=0
MOVL C01190 V=800.0 PL=0
MOVL C01191 V=800.0 PL=0
MOVL C01192 V=800.0 PL=0
MOVL C01193 V=800.0 PL=0
MOVL C01194 V=800.0 PL=0
MOVL C01195 V=800.0 PL=0
MOVL C01196 V=800.0 PL=0
MOVL C01197 V=800.0 PL=0
MOVL C01198 V=800.0 PL=0
MOVL C01199 V=800.0 PL=0
MOVL C01200 V=800.0 PL=0
MOVL C01201 V=800.0 PL=0
MOVL C01202 V=800.0 PL=0
MOVL C01203 V=800.0 PL=0
MOVL C01204 V=800.0 PL=0
MOVL C01205 V=800.0 PL=0
MOVL C01206 V=800.0 PL=0
MOVL C01207 V=800.0 PL=0
MOVL C01208 V=800.0 PL=0
MOVL C01209 V=800.0 PL=0
MOVL C01210 V=800.0 PL=0
MOVL C01211 V=800.0 PL=0
MOVL C01212 V=800.0 PL=0
MOVL C01213 V=800.0 PL=0
MOVL C01214 V=800.0 PL=0
MOVL C01215 V=800.0 PL=0
MOVL C01216 V=800.0 PL=0
MOVL C01217 V=800.0 PL=0
MOVL C01218 V=800.0 PL=0
MOVL C01219 V=800.0 PL=0
MOVL C01220 V=800.0 PL=0
MOVL C01221 V=800.0 PL=0
MOVL C01222 V=800.0 PL=0
MOVL C01223 V=800.0 PL=0
MOVL C01224 V=800.0 PL=0
MOVL C01225 V=800.0 PL=0
MOVL C01226 V=800.0 PL=0
MOVL C01227 V=800.0 PL=0
MOVL C01228 V=800.0 PL=0
MOVL C01229 V=800.0 PL=0
MOVL C01230 V=800.0 PL=0
MOVL C01231 V=800.0 PL=0
MOVL C01232 V=800.0 PL=0
MOVL C01233 V=800.0 PL=0
MOVL C01234 V=800.0 PL=0
MOVL C01235 V=800.0 PL=0
MOVL C01236 V=800.0 PL=0
MOVL C01237 V=800.0 PL=0
MOVL C01238 V=800.0 PL=0
MOVL C01239 V=800.0 PL=0
MOVL C01240 V=800.0 PL=0
MOVL C01241 V=800.0 PL=0
MOVL C01242 V=800.0 PL=0
MOVL C01243 V=800.0 PL=0
MOVL C01244 V=800.0 PL=0
MOVL C01245 V=800.0 PL=0
MOVL C01246 V=800.0 PL=0
MOVL C01247 V=800.0 PL=0
MOVL C01248 V=800.0 PL=0
MOVL C01249 V=800.0 PL=0
MOVL C01250 V=800.0 PL=0
MOVL C01251 V=800.0 PL=0
MOVL C01252 V=800.0 PL=0
MOVL C01253 V=800.0 PL=0
MOVL C01254 V=800.0 PL=0
MOVL C01255 V=800.0 PL=0
MOVL C01256 V=800.0 PL=0
MOVL C01257 V=800.0 PL=0
MOVL C01258 V=800.0 PL=0
MOVL C01259 V=800.0 PL=0
MOVL C01260 V=800.0 PL=0
MOVL C01261 V=800.0 PL=0
MOVL C01262 V=800.0 PL=0
MOVL C01263 V=800.0 PL=0
MOVL C01264 V=800.0 PL=0
MOVL C01265 V=800.0 PL=0
MOVL C01266 V=800.0 PL=0
MOVL C01267 V=800.0 PL=0
MOVL C01268 V=800.0 PL=0
MOVL C01269 V=800.0 PL=0
MOVL C01270 V=800.0 PL=0
MOVL C01271 V=800.0 PL=0
MOVL C01272 V=800.0 PL=0
MOVL C01273 V=800.0 PL=0
MOVL C01274 V=800.0 PL=0
MOVL C01275 V=800.0 PL=0
MOVL C01276 V=800.0 PL=0
MOVL C01277 V=800.0 PL=0
MOVL C01278 V=800.0 PL=0
MOVL C01279 V=800.0 PL=0
MOVL C01280 V=800.0 PL=0
MOVL C01281 V=800.0 PL=0
MOVL C01282 V=800.0 PL=0
MOVL C01283 V=800.0 PL=0
MOVL C01284 V=800.0 PL=0
MOVL C01285 V=800.0 PL=0
MOVL C01286 V=800.0 PL=0
MOVL C01287 V=800.0 PL=0
MOVL C01288 V=800.0 PL=0
MOVL C01289 V=800.0 PL=0
MOVL C01290 V=800.0 PL=0
MOVL C01291 V=800.0 PL=0
MOVL C01292 V=800.0 PL=0
MOVL C01293 V=800.0 PL=0
MOVL C01294 V=800.0 PL=0
MOVL C01295 V=800.0 PL=0
MOVL C01296 V=800.0 PL=0
MOVL C01297 V=800.0 PL=0
MOVL C01298 V=800.0 PL=0
MOVL C01299 V=800.0 PL=0
MOVL C01300 V=800.0 PL=0
MOVL C01301 V=800.0 PL=0
MOVL C01302 V=800.0 PL=0
MOVL C01303 V=800.0 PL=0
MOVL C01304 V=800.0 PL=0
MOVL C01305 V=800.0 PL=0
MOVL C01306 V=800.0 PL=0
MOVL C01307 V=800.0 PL=0
MOVL C01308 V=800.0 PL=0
MOVL C01309 V=800.0 PL=0
MOVL C01310 V=800.0 PL=0
MOVL C01311 V=800.0 PL=0
MOVL C01312 V=800.0 PL=0
MOVL C01313 V=800.0 PL=0
MOVL C01314 V=800.0 PL=0
MOVL C01315 V=800.0 PL=0
MOVL C01316 V=800.0 PL=0
MOVL C01317 V=800.0 PL=0
MOVL C01318 V=800.0 PL=0
MOVL C01319 V=800.0 PL=0
MOVL C01320 V=800.0 PL=0
MOVL C01321 V=800.0 PL=0
MOVL C01322 V=800.0 PL=0
MOVL C01323 V=800.0 PL=0
MOVL C01324 V=800.0 PL=0
MOVL C01325 V=800.0 PL=0
MOVL C01326 V=800.0 PL=0
MOVL C01327 V=800.0 PL=0
MOVL C01328 V=800.0 PL=0
MOVL C01329 V=800.0 PL=0
MOVL C01330 V=800.0 PL=0
MOVL C01331 V=800.0 PL=0
MOVL C01332 V=800.0 PL=0
MOVL C01333 V=800.0 PL=0
MOVL C01334 V=800.0 PL=0
MOVL C01335 V=800.0 PL=0
MOVL C01336 V=800.0 PL=0
MOVL C01337 V=800.0 PL=0
MOVL C01338 V=800.0 PL=0
MOVL C01339 V=800.0 PL=0
MOVL C01340 V=800.0 PL=0
MOVL C01341 V=800.0 PL=0
MOVL C01342 V=800.0 PL=0
MOVL C01343 V=800.0 PL=0
MOVL C01344 V=800.0 PL=0
MOVL C01345 V=800.0 PL=0
MOVL C01346 V=800.0 PL=0
MOVL C01347 V=800.0 PL=0
MOVL C01348 V=800.0 PL=0
MOVL C01349 V=800.0 PL=0
MOVL C01350 V=800.0 PL=0
MOVL C01351 V=800.0 PL=0
MOVL C01352 V=800.0 PL=0
MOVL C01353 V=800.0 PL=0
MOVL C01354 V=800.0 PL=0
MOVL C01355 V=800.0 PL=0
MOVL C01356 V=800.0 PL=0
MOVL C01357 V=800.0 PL=0
MOVL C01358 V=800.0 PL=0
MOVL C01359 V=800.0 PL=0
MOVL C01360 V=800.0 PL=0
MOVL C01361 V=800.0 PL=0
MOVL C01362 V=800.0 PL=0
MOVL C01363 V=800.0 PL=0
MOVL C01364 V=800.0 PL=0
MOVL C01365 V=800.0 PL=0
MOVL C01366 V=800.0 PL=0
MOVL C01367 V=800.0 PL=0
MOVL C01368 V=800.0 PL=0
MOVL C01369 V=800.0 PL=0
MOVL C01370 V=800.0 PL=0
MOVL C01371 V=800.0 PL=0
MOVL C01372 V=800.0 PL=0
MOVL C01373 V=800.0 PL=0
MOVL C01374 V=800.0 PL=0
MOVL C01375 V=800.0 PL=0
MOVL C01376 V=800.0 PL=0
MOVL C01377 V=800.0 PL=0
MOVL C01378 V=800.0 PL=0
MOVL C01379 V=800.0 PL=0
MOVL C01380 V=800.0 PL=0
MOVL C01381 V=800.0 PL=0
MOVL C01382 V=800.0 PL=0
MOVL C01383 V=800.0 PL=0
MOVL C01384 V=800.0 PL=0
MOVL C01385 V=800.0 PL=0
MOVL C01386 V=800.0 PL=0
MOVL C01387 V=800.0 PL=0
MOVL C01388 V=800.0 PL=0
MOVL C01389 V=800.0 PL=0
MOVL C01390 V=800.0 PL=0
MOVL C01391 V=800.0 PL=0
MOVL C01392 V=800.0 PL=0
MOVL C01393 V=800.0 PL=0
MOVL C01394 V=800.0 PL=0
MOVL C01395 V=800.0 PL=0
MOVL C01396 V=800.0 PL=0
MOVL C01397 V=800.0 PL=0
MOVL C01398 V=800.0 PL=0
MOVL C01399 V=800.0 PL=0
MOVL C01400 V=800.0 PL=0
MOVL C01401 V=800.0 PL=0
MOVL C01402 V=800.0 PL=0
MOVL C01403 V=800.0 PL=0
MOVL C01404 V=800.0 PL=0
MOVL C01405 V=800.0 PL=0
MOVL C01406 V=800.0 PL=0
MOVL C01407 V=800.0 PL=0
MOVL C01408 V=800.0 PL=0
MOVL C01409 V=800.0 PL=0
MOVL C01410 V=800.0 PL=0
MOVL C01411 V=800.0 PL=0
MOVL C01412 V=800.0 PL=0
MOVL C01413 V=800.0 PL=0
MOVL C01414 V=800.0 PL=0
MOVL C01415 V=800.0 PL=0
MOVL C01416 V=800.0 PL=0
MOVL C01417 V=800.0 PL=0
MOVL C01418 V=800.0 PL=0
MOVL C01419 V=800.0 PL=0
MOVL C01420 V=800.0 PL=0
MOVL C01421 V=800.0 PL=0
MOVL C01422 V=800.0 PL=0
MOVL C01423 V=800.0 PL=0
MOVL C01424 V=800.0 PL=0
MOVL C01425 V=800.0 PL=0
MOVL C01426 V=800.0 PL=0
MOVL C01427 V=800.0 PL=0
MOVL C01428 V=800.0 PL=0
MOVL C01429 V=800.0 PL=0
MOVL C01430 V=800.0 PL=0
MOVL C01431 V=800.0 PL=0
MOVL C01432 V=800.0 PL=0
MOVL C01433 V=800.0 PL=0
MOVL C01434 V=800.0 PL=0
MOVL C01435 V=800.0 PL=0
MOVL C01436 V=800.0 PL=0
MOVL C01437 V=800.0 PL=0
MOVL C01438 V=800.0 PL=0
MOVL C01439 V=800.0 PL=0
MOVL C01440 V=800.0 PL=0
MOVL C01441 V=800.0 PL=0
MOVL C01442 V=800.0 PL=0
MOVL C01443 V=800.0 PL=0
MOVL C01444 V=800.0 PL=0
MOVL C01445 V=800.0 PL=0
MOVL C01446 V=800.0 PL=0
MOVL C01447 V=800.0 PL=0
MOVL C01448 V=800.0 PL=0
MOVL C01449 V=800.0 PL=0
MOVL C01450 V=800.0 PL=0
MOVL C01451 V=800.0 PL=0
MOVL C01452 V=800.0 PL=0
MOVL C01453 V=800.0 PL=0
MOVL C01454 V=800.0 PL=0
MOVL C01455 V=800.0 PL=0
MOVL C01456 V=800.0 PL=0
MOVL C01457 V=800.0 PL=0
MOVL C01458 V=800.0 PL=0
MOVL C01459 V=800.0 PL=0
MOVL C01460 V=800.0 PL=0
MOVL C01461 V=800.0 PL=0
MOVL C01462 V=800.0 PL=0
MOVL C01463 V=800.0 PL=0
MOVL C01464 V=800.0 PL=0
MOVL C01465 V=800.0 PL=0
MOVL C01466 V=800.0 PL=0
MOVL C01467 V=800.0 PL=0
MOVL C01468 V=800.0 PL=0
MOVL C01469 V=800.0 PL=0
MOVL C01470 V=800.0 PL=0
MOVL C01471 V=800.0 PL=0
MOVL C01472 V=800.0 PL=0
MOVL C01473 V=800.0 PL=0
MOVL C01474 V=800.0 PL=0
MOVL C01475 V=800.0 PL=0
MOVL C01476 V=800.0 PL=0
MOVL C01477 V=800.0 PL=0
MOVL C01478 V=800.0 PL=0
MOVL C01479 V=800.0 PL=0
MOVL C01480 V=800.0 PL=0
MOVL C01481 V=800.0 PL=0
MOVL C01482 V=800.0 PL=0
MOVL C01483 V=800.0 PL=0
MOVL C01484 V=800.0 PL=0
MOVL C01485 V=800.0 PL=0
MOVL C01486 V=800.0 PL=0
MOVL C01487 V=800.0 PL=0
MOVL C01488 V=800.0 PL=0
MOVL C01489 V=800.0 PL=0
MOVL C01490 V=800.0 PL=0
MOVL C01491 V=800.0 PL=0
MOVL C01492 V=800.0 PL=0
MOVL C01493 V=800.0 PL=0
MOVL C01494 V=800.0 PL=0
MOVL C01495 V=800.0 PL=0
MOVL C01496 V=800.0 PL=0
MOVL C01497 V=800.0 PL=0
MOVL C01498 V=800.0 PL=0
MOVL C01499 V=800.0 PL=0
MOVL C01500 V=800.0 PL=0
MOVL C01501 V=800.0 PL=0
MOVL C01502 V=800.0 PL=0
MOVL C01503 V=800.0 PL=0
MOVL C01504 V=800.0 PL=0
MOVL C01505 V=800.0 PL=0
MOVL C01506 V=800.0 PL=0
MOVL C01507 V=800.0 PL=0
MOVL C01508 V=800.0 PL=0
MOVL C01509 V=800.0 PL=0
MOVL C01510 V=800.0 PL=0
MOVL C01511 V=800.0 PL=0
MOVL C01512 V=800.0 PL=0
MOVL C01513 V=800.0 PL=0
MOVL C01514 V=800.0 PL=0
MOVL C01515 V=800.0 PL=0
MOVL C01516 V=800.0 PL=0
MOVL C01517 V=800.0 PL=0
MOVL C01518 V=800.0 PL=0
MOVL C01519 V=800.0 PL=0
MOVL C01520 V=800.0 PL=0
MOVL C01521 V=800.0 PL=0
MOVL C01522 V=800.0 PL=0
MOVL C01523 V=800.0 PL=0
MOVL C01524 V=800.0 PL=0
MOVL C01525 V=800.0 PL=0
MOVL C01526 V=800.0 PL=0
MOVL C01527 V=800.0 PL=0
MOVL C01528 V=800.0 PL=0
MOVL C01529 V=800.0 PL=0
MOVL C01530 V=800.0 PL=0
MOVL C01531 V=800.0 PL=0
MOVL C01532 V=800.0 PL=0
MOVL C01533 V=800.0 PL=0
MOVL C01534 V=800.0 PL=0
MOVL C01535 V=800.0 PL=0
MOVL C01536 V=800.0 PL=0
MOVL C01537 V=800.0 PL=0
MOVL C01538 V=800.0 PL=0
MOVL C01539 V=800.0 PL=0
MOVL C01540 V=800.0 PL=0
MOVL C01541 V=800.0 PL=0
MOVL C01542 V=800.0 PL=0
MOVL C01543 V=800.0 PL=0
MOVL C01544 V=800.0 PL=0
MOVL C01545 V=800.0 PL=0
MOVL C01546 V=800.0 PL=0
MOVL C01547 V=800.0 PL=0
MOVL C01548 V=800.0 PL=0
MOVL C01549 V=800.0 PL=0
MOVL C01550 V=800.0 PL=0
MOVL C01551 V=800.0 PL=0
MOVL C01552 V=800.0 PL=0
MOVL C01553 V=800.0 PL=0
MOVL C01554 V=800.0 PL=0
MOVL C01555 V=800.0 PL=0
MOVL C01556 V=800.0 PL=0
MOVL C01557 V=800.0 PL=0
MOVL C01558 V=800.0 PL=0
MOVL C01559 V=800.0 PL=0
MOVL C01560 V=800.0 PL=0
MOVL C01561 V=800.0 PL=0
MOVL C01562 V=800.0 PL=0
MOVL C01563 V=800.0 PL=0
MOVL C01564 V=800.0 PL=0
MOVL C01565 V=800.0 PL=0
MOVL C01566 V=800.0 PL=0
MOVL C01567 V=800.0 PL=0
MOVL C01568 V=800.0 PL=0
MOVL C01569 V=800.0 PL=0
MOVL C01570 V=800.0 PL=0
MOVL C01571 V=800.0 PL=0
MOVL C01572 V=800.0 PL=0
MOVL C01573 V=800.0 PL=0
MOVL C01574 V=800.0 PL=0
MOVL C01575 V=800.0 PL=0
MOVL C01576 V=800.0 PL=0
MOVL C01577 V=800.0 PL=0
MOVL C01578 V=800.0 PL=0
MOVL C01579 V=800.0 PL=0
MOVL C01580 V=800.0 PL=0
MOVL C01581 V=800.0 PL=0
MOVL C01582 V=800.0 PL=0
MOVL C01583 V=800.0 PL=0
MOVL C01584 V=800.0 PL=0
MOVL C01585 V=800.0 PL=0
MOVL C01586 V=800.0 PL=0
MOVL C01587 V=800.0 PL=0
MOVL C01588 V=800.0 PL=0
MOVL C01589 V=800.0 PL=0
MOVL C01590 V=800.0 PL=0
MOVL C01591 V=800.0 PL=0
MOVL C01592 V=800.0 PL=0
MOVL C01593 V=800.0 PL=0
MOVL C01594 V=800.0 PL=0
MOVL C01595 V=800.0 PL=0
MOVL C01596 V=800.0 PL=0
MOVL C01597 V=800.0 PL=0
MOVL C01598 V=800.0 PL=0
MOVL C01599 V=800.0 PL=0
MOVL C01600 V=800.0 PL=0
MOVL C01601 V=800.0 PL=0
MOVL C01602 V=800.0 PL=0
MOVL C01603 V=800.0 PL=0
MOVL C01604 V=800.0 PL=0
MOVL C01605 V=800.0 PL=0
MOVL C01606 V=800.0 PL=0
MOVL C01607 V=800.0 PL=0
MOVL C01608 V=800.0 PL=0
MOVL C01609 V=800.0 PL=0
MOVL C01610 V=800.0 PL=0
MOVL C01611 V=800.0 PL=0
MOVL C01612 V=800.0 PL=0
MOVL C01613 V=800.0 PL=0
MOVL C01614 V=800.0 PL=0
MOVL C01615 V=800.0 PL=0
MOVL C01616 V=800.0 PL=0
MOVL C01617 V=800.0 PL=0
MOVL C01618 V=800.0 PL=0
MOVL C01619 V=800.0 PL=0
MOVL C01620 V=800.0 PL=0
MOVL C01621 V=800.0 PL=0
MOVL C01622 V=800.0 PL=0
MOVL C01623 V=800.0 PL=0
MOVL C01624 V=800.0 PL=0
MOVL C01625 V=800.0 PL=0
MOVL C01626 V=800.0 PL=0
MOVL C01627 V=800.0 PL=0
MOVL C01628 V=800.0 PL=0
MOVL C01629 V=800.0 PL=0
MOVL C01630 V=800.0 PL=0
MOVL C01631 V=800.0 PL=0
MOVL C01632 V=800.0 PL=0
MOVL C01633 V=800.0 PL=0
MOVL C01634 V=800.0 PL=0
MOVL C01635 V=800.0 PL=0
MOVL C01636 V=800.0 PL=0
MOVL C01637 V=800.0 PL=0
MOVL C01638 V=800.0 PL=0
MOVL C01639 V=800.0 PL=0
MOVL C01640 V=800.0 PL=0
MOVL C01641 V=800.0 PL=0
MOVL C01642 V=800.0 PL=0
MOVL C01643 V=800.0 PL=0
MOVL C01644 V=800.0 PL=0
MOVL C01645 V=800.0 PL=0
MOVL C01646 V=800.0 PL=0
MOVL C01647 V=800.0 PL=0
MOVL C01648 V=800.0 PL=0
MOVL C01649 V=800.0 PL=0
MOVL C01650 V=800.0 PL=0
MOVL C01651 V=800.0 PL=0
MOVL C01652 V=800.0 PL=0
MOVL C01653 V=800.0 PL=0
MOVL C01654 V=800.0 PL=0
MOVL C01655 V=800.0 PL=0
MOVL C01656 V=800.0 PL=0
MOVL C01657 V=800.0 PL=0
MOVL C01658 V=800.0 PL=0
MOVL C01659 V=800.0 PL=0
MOVL C01660 V=800.0 PL=0
MOVL C01661 V=800.0 PL=0
MOVL C01662 V=800.0 PL=0
MOVL C01663 V=800.0 PL=0
MOVL C01664 V=800.0 PL=0
MOVL C01665 V=800.0 PL=0
MOVL C01666 V=800.0 PL=0
MOVL C01667 V=800.0 PL=0
MOVL C01668 V=800.0 PL=0
MOVL C01669 V=800.0 PL=0
MOVL C01670 V=800.0 PL=0
MOVL C01671 V=800.0 PL=0
MOVL C01672 V=800.0 PL=0
MOVL C01673 V=800.0 PL=0
MOVL C01674 V=800.0 PL=0
MOVL C01675 V=800.0 PL=0
MOVL C01676 V=800.0 PL=0
MOVL C01677 V=800.0 PL=0
MOVL C01678 V=800.0 PL=0
MOVL C01679 V=800.0 PL=0
MOVL C01680 V=800.0 PL=0
MOVL C01681 V=800.0 PL=0
MOVL C01682 V=800.0 PL=0
MOVL C01683 V=800.0 PL=0
MOVL C01684 V=800.0 PL=0
MOVL C01685 V=800.0 PL=0
MOVL C01686 V=800.0 PL=0
MOVL C01687 V=800.0 PL=0
MOVL C01688 V=800.0 PL=0
MOVL C01689 V=800.0 PL=0
MOVL C01690 V=800.0 PL=0
MOVL C01691 V=800.0 PL=0
MOVL C01692 V=800.0 PL=0
MOVL C01693 V=800.0 PL=0
MOVL C01694 V=800.0 PL=0
MOVL C01695 V=800.0 PL=0
MOVL C01696 V=800.0 PL=0
MOVL C01697 V=800.0 PL=0
MOVL C01698 V=800.0 PL=0
MOVL C01699 V=800.0 PL=0
MOVL C01700 V=800.0 PL=0
MOVL C01701 V=800.0 PL=0
MOVL C01702 V=800.0 PL=0
MOVL C01703 V=800.0 PL=0
MOVL C01704 V=800.0 PL=0
MOVL C01705 V=800.0 PL=0
MOVL C01706 V=800.0 PL=0
MOVL C01707 V=800.0 PL=0
MOVL C01708 V=800.0 PL=0
MOVL C01709 V=800.0 PL=0
MOVL C01710 V=800.0 PL=0
MOVL C01711 V=800.0 PL=0
MOVL C01712 V=800.0 PL=0
MOVL C01713 V=800.0 PL=0
MOVL C01714 V=800.0 PL=0
MOVL C01715 V=800.0 PL=0
MOVL C01716 V=800.0 PL=0
MOVL C01717 V=800.0 PL=0
MOVL C01718 V=800.0 PL=0
MOVL C01719 V=800.0 PL=0
MOVL C01720 V=800.0 PL=0
MOVL C01721 V=800.0 PL=0
MOVL C01722 V=800.0 PL=0
MOVL C01723 V=800.0 PL=0
MOVL C01724 V=800.0 PL=0
MOVL C01725 V=800.0 PL=0
MOVL C01726 V=800.0 PL=0
MOVL C01727 V=800.0 PL=0
MOVL C01728 V=800.0 PL=0
MOVL C01729 V=800.0 PL=0
MOVL C01730 V=800.0 PL=0
MOVL C01731 V=800.0 PL=0
MOVL C01732 V=800.0 PL=0
MOVL C01733 V=800.0 PL=0
MOVL C01734 V=800.0 PL=0
MOVL C01735 V=800.0 PL=0
MOVL C01736 V=800.0 PL=0
MOVL C01737 V=800.0 PL=0
MOVL C01738 V=800.0 PL=0
MOVL C01739 V=800.0 PL=0
MOVL C01740 V=800.0 PL=0
MOVL C01741 V=800.0 PL=0
MOVL C01742 V=800.0 PL=0
MOVL C01743 V=800.0 PL=0
MOVL C01744 V=800.0 PL=0
MOVL C01745 V=800.0 PL=0
MOVL C01746 V=800.0 PL=0
MOVL C01747 V=800.0 PL=0
MOVL C01748 V=800.0 PL=0
MOVL C01749 V=800.0 PL=0
MOVL C01750 V=800.0 PL=0
MOVL C01751 V=800.0 PL=0
MOVL C01752 V=800.0 PL=0
MOVL C01753 V=800.0 PL=0
MOVL C01754 V=800.0 PL=0
MOVL C01755 V=800.0 PL=0
MOVL C01756 V=800.0 PL=0
MOVL C01757 V=800.0 PL=0
MOVL C01758 V=800.0 PL=0
MOVL C01759 V=800.0 PL=0
MOVL C01760 V=800.0 PL=0
MOVL C01761 V=800.0 PL=0
MOVL C01762 V=800.0 PL=0
MOVL C01763 V=800.0 PL=0
MOVL C01764 V=800.0 PL=0
MOVL C01765 V=800.0 PL=0
MOVL C01766 V=800.0 PL=0
MOVL C01767 V=800.0 PL=0
MOVL C01768 V=800.0 PL=0
MOVL C01769 V=800.0 PL=0
MOVL C01770 V=800.0 PL=0
MOVL C01771 V=800.0 PL=0
MOVL C01772 V=800.0 PL=0
MOVL C01773 V=800.0 PL=0
MOVL C01774 V=800.0 PL=0
MOVL C01775 V=800.0 PL=0
MOVL C01776 V=800.0 PL=0
MOVL C01777 V=800.0 PL=0
MOVL C01778 V=800.0 PL=0
MOVL C01779 V=800.0 PL=0
MOVL C01780 V=800.0 PL=0
MOVL C01781 V=800.0 PL=0
MOVL C01782 V=800.0 PL=0
MOVL C01783 V=800.0 PL=0
MOVL C01784 V=800.0 PL=0
MOVL C01785 V=800.0 PL=0
MOVL C01786 V=800.0 PL=0
MOVL C01787 V=800.0 PL=0
MOVL C01788 V=800.0 PL=0
MOVL C01789 V=800.0 PL=0
MOVL C01790 V=800.0 PL=0
MOVL C01791 V=800.0 PL=0
MOVL C01792 V=800.0 PL=0
MOVL C01793 V=800.0 PL=0
MOVL C01794 V=800.0 PL=0
MOVL C01795 V=800.0 PL=0
MOVL C01796 V=800.0 PL=0
MOVL C01797 V=800.0 PL=0
MOVL C01798 V=800.0 PL=0
MOVL C01799 V=800.0 PL=0
MOVL C01800 V=800.0 PL=0
MOVL C01801 V=800.0 PL=0
MOVL C01802 V=800.0 PL=0
MOVL C01803 V=800.0 PL=0
MOVL C01804 V=800.0 PL=0
MOVL C01805 V=800.0 PL=0
MOVL C01806 V=800.0 PL=0
MOVL C01807 V=800.0 PL=0
MOVL C01808 V=800.0 PL=0
MOVL C01809 V=800.0 PL=0
MOVL C01810 V=800.0 PL=0
MOVL C01811 V=800.0 PL=0
MOVL C01812 V=800.0 PL=0
MOVL C01813 V=800.0 PL=0
MOVL C01814 V=800.0 PL=0
MOVL C01815 V=800.0 PL=0
MOVL C01816 V=800.0 PL=0
MOVL C01817 V=800.0 PL=0
MOVL C01818 V=800.0 PL=0
MOVL C01819 V=800.0 PL=0
MOVL C01820 V=800.0 PL=0
MOVL C01821 V=800.0 PL=0
MOVL C01822 V=800.0 PL=0
MOVL C01823 V=800.0 PL=0
MOVL C01824 V=800.0 PL=0
MOVL C01825 V=800.0 PL=0
MOVL C01826 V=800.0 PL=0
MOVL C01827 V=800.0 PL=0
MOVL C01828 V=800.0 PL=0
MOVL C01829 V=800.0 PL=0
MOVL C01830 V=800.0 PL=0
MOVL C01831 V=800.0 PL=0
MOVL C01832 V=800.0 PL=0
MOVL C01833 V=800.0 PL=0
MOVL C01834 V=800.0 PL=0
MOVL C01835 V=800.0 PL=0
MOVL C01836 V=800.0 PL=0
MOVL C01837 V=800.0 PL=0
MOVL C01838 V=800.0 PL=0
MOVL C01839 V=800.0 PL=0
MOVL C01840 V=800.0 PL=0
MOVL C01841 V=800.0 PL=0
MOVL C01842 V=800.0 PL=0
MOVL C01843 V=800.0 PL=0
MOVL C01844 V=800.0 PL=0
MOVL C01845 V=800.0 PL=0
MOVL C01846 V=800.0 PL=0
MOVL C01847 V=800.0 PL=0
MOVL C01848 V=800.0 PL=0
MOVL C01849 V=800.0 PL=0
MOVL C01850 V=800.0 PL=0
MOVL C01851 V=800.0 PL=0
MOVL C01852 V=800.0 PL=0
MOVL C01853 V=800.0 PL=0
MOVL C01854 V=800.0 PL=0
MOVL C01855 V=800.0 PL=0
MOVL C01856 V=800.0 PL=0
MOVL C01857 V=800.0 PL=0
MOVL C01858 V=800.0 PL=0
MOVL C01859 V=800.0 PL=0
MOVL C01860 V=800.0 PL=0
MOVL C01861 V=800.0 PL=0
MOVL C01862 V=800.0 PL=0
MOVL C01863 V=800.0 PL=0
MOVL C01864 V=800.0 PL=0
MOVL C01865 V=800.0 PL=0
MOVL C01866 V=800.0 PL=0
MOVL C01867 V=800.0 PL=0
MOVL C01868 V=800.0 PL=0
MOVL C01869 V=800.0 PL=0
MOVL C01870 V=800.0 PL=0
MOVL C01871 V=800.0 PL=0
MOVL C01872 V=800.0 PL=0
MOVL C01873 V=800.0 PL=0
MOVL C01874 V=800.0 PL=0
MOVL C01875 V=800.0 PL=0
MOVL C01876 V=800.0 PL=0
MOVL C01877 V=800.0 PL=0
MOVL C01878 V=800.0 PL=0
MOVL C01879 V=800.0 PL=0
MOVL C01880 V=800.0 PL=0
MOVL C01881 V=800.0 PL=0
MOVL C01882 V=800.0 PL=0
MOVL C01883 V=800.0 PL=0
MOVL C01884 V=800.0 PL=0
MOVL C01885 V=800.0 PL=0
MOVL C01886 V=800.0 PL=0
MOVL C01887 V=800.0 PL=0
MOVL C01888 V=800.0 PL=0
MOVL C01889 V=800.0 PL=0
MOVL C01890 V=800.0 PL=0
MOVL C01891 V=800.0 PL=0
MOVL C01892 V=800.0 PL=0
MOVL C01893 V=800.0 PL=0
MOVL C01894 V=800.0 PL=0
MOVL C01895 V=800.0 PL=0
MOVL C01896 V=800.0 PL=0
MOVL C01897 V=800.0 PL=0
MOVL C01898 V=800.0 PL=0
MOVL C01899 V=800.0 PL=0
MOVL C01900 V=800.0 PL=0
MOVL C01901 V=800.0 PL=0
MOVL C01902 V=800.0 PL=0
MOVL C01903 V=800.0 PL=0
MOVL C01904 V=800.0 PL=0
MOVL C01905 V=800.0 PL=0
MOVL C01906 V=800.0 PL=0
MOVL C01907 V=800.0 PL=0
MOVL C01908 V=800.0 PL=0
MOVL C01909 V=800.0 PL=0
MOVL C01910 V=800.0 PL=0
MOVL C01911 V=800.0 PL=0
MOVL C01912 V=800.0 PL=0
MOVL C01913 V=800.0 PL=0
MOVL C01914 V=800.0 PL=0
MOVL C01915 V=800.0 PL=0
MOVL C01916 V=800.0 PL=0
MOVL C01917 V=800.0 PL=0
MOVL C01918 V=800.0 PL=0
MOVL C01919 V=800.0 PL=0
MOVL C01920 V=800.0 PL=0
MOVL C01921 V=800.0 PL=0
MOVL C01922 V=800.0 PL=0
MOVL C01923 V=800.0 PL=0
MOVL C01924 V=800.0 PL=0
MOVL C01925 V=800.0 PL=0
MOVL C01926 V=800.0 PL=0
MOVL C01927 V=800.0 PL=0
MOVL C01928 V=800.0 PL=0
MOVL C01929 V=800.0 PL=0
MOVL C01930 V=800.0 PL=0
MOVL C01931 V=800.0 PL=0
MOVL C01932 V=800.0 PL=0
MOVL C01933 V=800.0 PL=0
MOVL C01934 V=800.0 PL=0
MOVL C01935 V=800.0 PL=0
MOVL C01936 V=800.0 PL=0
MOVL C01937 V=800.0 PL=0
MOVL C01938 V=800.0 PL=0
MOVL C01939 V=800.0 PL=0
MOVL C01940 V=800.0 PL=0
MOVL C01941 V=800.0 PL=0
MOVL C01942 V=800.0 PL=0
MOVL C01943 V=800.0 PL=0
MOVL C01944 V=800.0 PL=0
MOVL C01945 V=800.0 PL=0
MOVL C01946 V=800.0 PL=0
MOVL C01947 V=800.0 PL=0
MOVL C01948 V=800.0 PL=0
MOVL C01949 V=800.0 PL=0
MOVL C01950 V=800.0 PL=0
MOVL C01951 V=800.0 PL=0
MOVL C01952 V=800.0 PL=0
MOVL C01953 V=800.0 PL=0
MOVL C01954 V=800.0 PL=0
MOVL C01955 V=800.0 PL=0
MOVL C01956 V=800.0 PL=0
MOVL C01957 V=800.0 PL=0
MOVL C01958 V=800.0 PL=0
MOVL C01959 V=800.0 PL=0
MOVL C01960 V=800.0 PL=0
MOVL C01961 V=800.0 PL=0
MOVL C01962 V=800.0 PL=0
MOVL C01963 V=800.0 PL=0
MOVL C01964 V=800.0 PL=0
MOVL C01965 V=800.0 PL=0
MOVL C01966 V=800.0 PL=0
MOVL C01967 V=800.0 PL=0
MOVL C01968 V=800.0 PL=0
MOVL C01969 V=800.0 PL=0
MOVL C01970 V=800.0 PL=0
MOVL C01971 V=800.0 PL=0
MOVL C01972 V=800.0 PL=0
MOVL C01973 V=800.0 PL=0
MOVL C01974 V=800.0 PL=0
MOVL C01975 V=800.0 PL=0
MOVL C01976 V=800.0 PL=0
MOVL C01977 V=800.0 PL=0
MOVL C01978 V=800.0 PL=0
MOVL C01979 V=800.0 PL=0
MOVL C01980 V=800.0 PL=0
MOVL C01981 V=800.0 PL=0
MOVL C01982 V=800.0 PL=0
MOVL C01983 V=800.0 PL=0
MOVL C01984 V=800.0 PL=0
MOVL C01985 V=800.0 PL=0
MOVL C01986 V=800.0 PL=0
MOVL C01987 V=800.0 PL=0
MOVL C01988 V=800.0 PL=0
MOVL C01989 V=800.0 PL=0
MOVL C01990 V=800.0 PL=0
MOVL C01991 V=800.0 PL=0
MOVL C01992 V=800.0 PL=0
MOVL C01993 V=800.0 PL=0
MOVL C01994 V=800.0 PL=0
MOVL C01995 V=800.0 PL=0
MOVL C01996 V=800.0 PL=0
MOVL C01997 V=800.0 PL=0
MOVL C01998 V=800.0 PL=0
MOVL C01999 V=800.0 PL=0
MOVL C02000 V=800.0 PL=0
MOVL C02001 V=800.0 PL=0
MOVL C02002 V=800.0 PL=0
MOVL C02003 V=800.0 PL=0
MOVL C02004 V=800.0 PL=0
MOVL C02005 V=800.0 PL=0
MOVL C02006 V=800.0 PL=0
MOVL C02007 V=800.0 PL=0
MOVL C02008 V=800.0 PL=0
MOVL C02009 V=800.0 PL=0
MOVL C02010 V=800.0 PL=0
MOVL C02011 V=800.0 PL=0
MOVL C02012 V=800.0 PL=0
MOVL C02013 V=800.0 PL=0
MOVL C02014 V=800.0 PL=0
MOVL C02015 V=800.0 PL=0
MOVL C02016 V=800.0 PL=0
MOVL C02017 V=800.0 PL=0
MOVL C02018 V=800.0 PL=0
MOVL C02019 V=800.0 PL=0
MOVL C02020 V=800.0 PL=0
MOVL C02021 V=800.0 PL=0
MOVL C02022 V=800.0 PL=0
